C01815=1065.193,415.285,383.687,175.579,36.944,156.981
C01816=1065.183,414.985,383.742,175.571,36.933,156.978
C01817=1065.173,414.684,383.796,175.562,36.921,156.975
C01818=1065.163,414.383,383.850,175.554,36.909,156.972
C01819=1065.153,414.082,383.904,175.545,36.897,156.969
C01820=1065.144,413.837,383.948,175.539,36.887,156.967
C01821=1065.136,413.591,383.993,175.532,36.878,156.964
C01822=1065.128,413.345,384.036,175.525,36.869,156.962
C01823=1065.120,413.099,384.080,175.519,36.859,156.960
C01824=1065.111,412.853,384.125,175.511,36.850,156.957
C01825=1065.103,412.606,384.168,175.505,36.840,156.955
C01826=1065.095,412.361,384.213,175.498,36.831,156.952
C01827=1065.086,412.115,384.256,175.492,36.822,156.950
C01828=1065.079,411.869,384.300,175.485,36.812,156.948
C01829=1065.071,411.623,384.344,175.479,36.803,156.945
C01830=1065.063,411.377,384.388,175.472,36.794,156.943
C01831=1065.054,411.131,384.432,175.466,36.784,156.941
C01832=1065.046,410.885,384.475,175.459,36.775,156.938
C01833=1065.039,410.639,384.519,175.452,36.766,156.936
C01834=1065.030,410.393,384.563,175.445,36.756,156.934
C01835=1065.022,410.147,384.606,175.439,36.747,156.931
C01836=1065.014,409.900,384.650,175.432,36.738,156.929
C01837=1065.006,409.654,384.693,175.426,36.729,156.927
C01838=1064.998,409.409,384.737,175.420,36.720,156.924
C01839=1064.991,409.163,384.780,175.413,36.711,156.922
C01840=1064.983,408.917,384.824,175.407,36.702,156.920
C01841=1064.974,408.671,384.867,175.400,36.693,156.918
C01842=1064.966,408.424,384.911,175.394,36.684,156.915
C01843=1064.959,408.178,384.954,175.388,36.675,156.913
C01844=1064.951,407.932,384.997,175.381,36.666,156.911
C01845=1064.943,407.686,385.041,175.376,36.657,156.909
C01846=1064.935,407.440,385.084,175.369,36.648,156.906
C01847=1064.927,407.194,385.127,175.363,36.639,156.904
C01848=1064.920,406.948,385.171,175.357,36.630,156.902
C01849=1064.912,406.702,385.214,175.350,36.621,156.900
C01850=1064.903,406.456,385.257,175.344,36.613,156.898
C01851=1064.896,406.210,385.300,175.338,36.603,156.895
C01852=1064.888,405.963,385.343,175.331,36.595,156.893
C01853=1064.880,405.717,385.386,175.325,36.586,156.891
C01854=1064.872,405.471,385.429,175.320,36.577,156.889
C01855=1064.865,405.225,385.472,175.313,36.568,156.887
C01856=1064.856,404.978,385.515,175.307,36.560,156.885
C01857=1064.850,404.732,385.558,175.301,36.551,156.882
C01858=1064.841,404.486,385.601,175.295,36.543,156.880
C01859=1064.833,404.240,385.644,175.288,36.534,156.878
C01860=1064.826,403.994,385.686,175.283,36.525,156.876
C01861=1064.817,403.748,385.729,175.277,36.517,156.874
C01862=1064.810,403.501,385.772,175.270,36.508,156.872
C01863=1064.802,403.255,385.814,175.264,36.500,156.870
C01864=1064.794,403.009,385.857,175.258,36.492,156.868
C01865=1064.787,402.762,385.900,175.253,36.483,156.866
C01866=1064.779,402.516,385.941,175.247,36.474,156.863
C01867=1064.771,402.270,385.985,175.240,36.466,156.861
C01868=1064.763,402.023,386.027,175.234,36.458,156.859
C01869=1064.756,401.777,386.069,175.229,36.449,156.857
C01870=1064.748,401.531,386.111,175.223,36.441,156.855
C01871=1064.740,401.285,386.154,175.217,36.433,156.853
C01872=1064.730,400.989,386.205,175.210,36.422,156.851
C01873=1064.721,400.693,386.256,175.203,36.413,156.848
C01874=1064.712,400.397,386.307,175.195,36.403,156.846
C01875=1064.703,400.101,386.357,175.189,36.393,156.843
C01876=1064.695,399.854,386.400,175.183,36.385,156.841
C01877=1064.688,399.608,386.441,175.177,36.376,156.839
C01878=1064.680,399.362,386.483,175.171,36.368,156.838
C01879=1064.672,399.116,386.526,175.165,36.360,156.836
C01880=1064.664,398.870,386.568,175.159,36.352,156.834
C01881=1064.657,398.624,386.610,175.154,36.344,156.832
C01882=1064.649,398.377,386.653,175.148,36.336,156.830
C01883=1064.642,398.130,386.694,175.143,36.328,156.828
C01884=1064.634,397.884,386.736,175.137,36.320,156.826
C01885=1064.627,397.638,386.778,175.131,36.312,156.824
C01886=1064.619,397.391,386.819,175.125,36.304,156.822
C01887=1064.611,397.145,386.861,175.119,36.296,156.820
C01888=1064.604,396.899,386.903,175.114,36.288,156.818
C01889=1064.596,396.652,386.944,175.108,36.280,156.816
C01890=1064.589,396.406,386.986,175.103,36.272,156.814
C01891=1064.581,396.160,387.028,175.097,36.264,156.812
C01892=1064.573,395.913,387.070,175.091,36.256,156.810
C01893=1064.566,395.667,387.112,175.086,36.248,156.808
C01894=1064.558,395.421,387.152,175.080,36.241,156.807
C01895=1064.550,395.174,387.194,175.075,36.233,156.805
C01896=1064.543,394.928,387.236,175.069,36.225,156.803
C01897=1064.536,394.682,387.277,175.064,36.217,156.801
C01898=1064.528,394.436,387.319,175.058,36.209,156.799
C01899=1064.521,394.189,387.360,175.053,36.202,156.797
C01900=1064.513,393.943,387.401,175.047,36.194,156.795
C01901=1064.506,393.697,387.443,175.042,36.186,156.793
C01902=1064.498,393.450,387.484,175.036,36.179,156.792
C01903=1064.490,393.204,387.525,175.031,36.171,156.790
C01904=1064.483,392.957,387.566,175.025,36.163,156.788
C01905=1064.476,392.711,387.607,175.020,36.156,156.786
C01906=1064.468,392.465,387.649,175.014,36.148,156.784
C01907=1064.460,392.218,387.690,175.009,36.141,156.782
C01908=1064.453,391.972,387.731,175.003,36.133,156.781
C01909=1064.446,391.725,387.773,174.998,36.125,156.779
C01910=1064.438,391.479,387.813,174.992,36.118,156.777
C01911=1064.430,391.232,387.854,174.987,36.110,156.775
C01912=1064.424,390.986,387.895,174.982,36.103,156.773
C01913=1064.416,390.740,387.936,174.976,36.095,156.772
C01914=1064.408,390.493,387.977,174.971,36.088,156.770
C01915=1064.401,390.247,388.018,174.965,36.080,156.768
C01916=1064.393,390.000,388.058,174.960,36.073,156.766
C01917=1064.386,389.753,388.099,174.954,36.066,156.765
C01918=1064.378,389.507,388.140,174.949,36.058,156.763
C01919=1064.371,389.261,388.181,174.944,36.051,156.761
C01920=1064.364,389.014,388.221,174.938,36.044,156.759
C01921=1064.356,388.768,388.262,174.933,36.037,156.758
C01922=1064.348,388.521,388.303,174.929,36.029,156.756
C01923=1064.341,388.274,388.343,174.923,36.022,156.754
C01924=1064.334,388.029,388.384,174.918,36.015,156.752
C01925=1064.326,387.782,388.424,174.912,36.007,156.751
C01926=1064.319,387.535,388.465,174.907,36.000,156.749
C01927=1064.311,387.289,388.505,174.902,35.993,156.747
C01928=1064.303,387.010,388.551,174.896,35.985,156.745
C01929=1064.295,386.730,388.597,174.890,35.977,156.743
C01930=1064.286,386.451,388.643,174.884,35.968,156.742
C01931=1064.278,386.171,388.689,174.878,35.961,156.740
C01932=1064.271,385.924,388.729,174.873,35.954,156.738
C01933=1064.264,385.677,388.769,174.868,35.946,156.736
C01934=1064.256,385.431,388.810,174.862,35.939,156.735
C01935=1064.249,385.185,388.849,174.858,35.932,156.733
C01936=1064.242,384.938,388.890,174.853,35.925,156.731
C01937=1064.234,384.692,388.930,174.847,35.918,156.730
C01938=1064.227,384.445,388.970,174.842,35.911,156.728
C01939=1064.220,384.198,389.011,174.837,35.904,156.726
C01940=1064.212,383.952,389.050,174.832,35.897,156.725
C01941=1064.205,383.704,389.091,174.827,35.890,156.723
C01942=1064.198,383.459,389.131,174.822,35.883,156.721
C01943=1064.190,383.212,389.171,174.817,35.876,156.720
C01944=1064.184,382.965,389.211,174.812,35.869,156.718
C01945=1064.176,382.718,389.251,174.807,35.862,156.717
C01946=1064.169,382.472,389.290,174.801,35.855,156.715
C01947=1064.162,382.225,389.331,174.797,35.848,156.713
C01948=1064.155,381.979,389.371,174.792,35.841,156.712
C01949=1064.147,381.732,389.410,174.787,35.834,156.710
C01950=1064.141,381.485,389.451,174.782,35.827,156.708
C01951=1064.134,381.239,389.490,174.776,35.821,156.707
C01952=1064.126,380.992,389.530,174.772,35.814,156.705
C01953=1064.119,380.746,389.569,174.767,35.807,156.704
C01954=1064.112,380.498,389.609,174.762,35.800,156.702
C01955=1064.105,380.252,389.649,174.757,35.794,156.701
C01956=1064.097,380.005,389.689,174.753,35.787,156.699
C01957=1064.090,379.759,389.728,174.747,35.780,156.697
C01958=1064.083,379.511,389.768,174.742,35.774,156.696
C01959=1064.076,379.265,389.807,174.737,35.767,156.694
C01960=1064.069,379.019,389.847,174.733,35.760,156.693
C01961=1064.061,378.772,389.886,174.728,35.754,156.691
C01962=1064.054,378.525,389.926,174.723,35.747,156.690
C01963=1064.047,378.278,389.965,174.718,35.740,156.688
C01964=1064.040,378.032,390.004,174.713,35.734,156.687
C01965=1064.033,377.785,390.043,174.708,35.727,156.685
C01966=1064.025,377.538,390.083,174.703,35.720,156.684
C01967=1064.018,377.291,390.122,174.698,35.714,156.682
C01968=1064.011,377.045,390.161,174.694,35.707,156.680
C01969=1064.004,376.798,390.200,174.689,35.701,156.679
C01970=1063.997,376.551,390.240,174.684,35.694,156.678
C01971=1063.990,376.304,390.279,174.680,35.688,156.676
C01972=1063.983,376.058,390.319,174.675,35.681,156.674
C01973=1063.976,375.811,390.357,174.670,35.675,156.673
C01974=1063.968,375.564,390.397,174.665,35.668,156.672
C01975=1063.961,375.318,390.436,174.660,35.661,156.670
C01976=1063.955,375.071,390.475,174.655,35.655,156.669
C01977=1063.948,374.824,390.514,174.650,35.649,156.667
C01978=1063.941,374.577,390.553,174.646,35.642,156.666
C01979=1063.933,374.330,390.592,174.641,35.636,156.664
C01980=1063.926,374.083,390.631,174.636,35.630,156.663
C01981=1063.919,373.837,390.670,174.632,35.623,156.661
C01982=1063.912,373.590,390.708,174.627,35.617,156.660
C01983=1063.905,373.343,390.747,174.622,35.610,156.658
C01984=1063.898,373.094,390.787,174.618,35.604,156.657
C01985=1063.892,372.845,390.826,174.613,35.597,156.655
C01986=1063.884,372.597,390.865,174.608,35.591,156.654
C01987=1063.877,372.347,390.904,174.604,35.584,156.652
C01988=1063.870,372.101,390.943,174.599,35.578,156.651
C01989=1063.863,371.854,390.981,174.594,35.572,156.650
C01990=1063.856,371.607,391.020,174.590,35.566,156.648
C01991=1063.849,371.360,391.059,174.585,35.560,156.647
C01992=1063.841,371.113,391.098,174.580,35.554,156.645
C01993=1063.835,370.866,391.136,174.576,35.548,156.644
C01994=1063.827,370.619,391.174,174.571,35.541,156.643
C01995=1063.820,370.372,391.213,174.566,35.535,156.641
C01996=1063.813,370.126,391.252,174.562,35.529,156.640
C01997=1063.806,369.878,391.289,174.557,35.522,156.638
C01998=1063.799,369.632,391.328,174.553,35.517,156.637
C01999=1063.792,369.385,391.367,174.549,35.511,156.635
C02000=1063.785,369.138,391.405,174.544,35.504,156.634
C02001=1063.778,368.891,391.443,174.540,35.498,156.633
C02002=1063.771,368.644,391.481,174.535,35.492,156.631
C02003=1063.764,368.397,391.520,174.530,35.486,156.630
C02004=1063.758,368.150,391.558,174.526,35.480,156.629
C02005=1063.750,367.904,391.597,174.521,35.474,156.627
C02006=1063.744,367.656,391.635,174.517,35.468,156.626
C02007=1063.736,367.410,391.673,174.512,35.462,156.624
C02008=1063.730,367.163,391.711,174.507,35.456,156.623
C02009=1063.723,366.916,391.750,174.503,35.449,156.622
C02010=1063.716,366.669,391.787,174.499,35.443,156.620
C02011=1063.710,366.421,391.825,174.495,35.438,156.619
C02012=1063.702,366.175,391.863,174.490,35.431,156.618
C02013=1063.695,365.928,391.902,174.485,35.425,156.616
C02014=1063.688,365.681,391.940,174.481,35.420,156.615
C02015=1063.682,365.434,391.978,174.476,35.413,156.614
C02016=1063.675,365.187,392.015,174.472,35.408,156.612
C02017=1063.668,364.940,392.054,174.468,35.402,156.611
C02018=1063.661,364.693,392.092,174.464,35.395,156.609
C02019=1063.654,364.446,392.130,174.459,35.390,156.608
C02020=1063.648,364.199,392.167,174.454,35.384,156.607
C02021=1063.641,363.952,392.205,174.450,35.378,156.606
C02022=1063.633,363.705,392.243,174.445,35.372,156.604
C02023=1063.627,363.458,392.281,174.442,35.366,156.603
C02024=1063.620,363.211,392.319,174.437,35.361,156.602
C02025=1063.612,362.964,392.356,174.433,35.355,156.600
C02026=1063.607,362.717,392.394,174.428,35.349,156.599
C02027=1063.599,362.470,392.432,174.424,35.343,156.598
C02028=1063.592,362.223,392.469,174.419,35.337,156.596
C02029=1063.585,361.975,392.507,174.416,35.332,156.595
C02030=1063.579,361.729,392.544,174.411,35.326,156.594
C02031=1063.572,361.482,392.582,174.406,35.320,156.593
C02032=1063.564,361.234,392.619,174.402,35.314,156.591
C02033=1063.557,360.987,392.657,174.398,35.309,156.590
C02034=1063.551,360.741,392.695,174.394,35.303,156.589
C02035=1063.544,360.493,392.732,174.389,35.297,156.588
C02036=1063.538,360.254,392.768,174.385,35.292,156.586
C02037=1063.531,360.015,392.804,174.381,35.286,156.585
C02038=1063.524,359.776,392.840,174.377,35.280,156.584
C02039=1063.518,359.537,392.876,174.372,35.275,156.583
C02040=1063.511,359.298,392.912,174.369,35.270,156.581
C02041=1063.505,359.059,392.949,174.364,35.264,156.580
C02042=1063.498,358.820,392.985,174.361,35.259,156.579
C02043=1063.491,358.581,393.021,174.356,35.253,156.578
C02044=1063.485,358.334,393.058,174.352,35.247,156.576
C02045=1063.478,358.087,393.095,174.348,35.242,156.575
C02046=1063.471,357.840,393.133,174.344,35.236,156.574
C02047=1063.464,357.592,393.169,174.339,35.230,156.573
C02048=1063.457,357.345,393.207,174.335,35.225,156.572
C02049=1063.451,357.098,393.243,174.331,35.220,156.570
C02050=1063.443,356.851,393.281,174.327,35.214,156.569
C02051=1063.437,356.604,393.317,174.322,35.208,156.568
C02052=1063.430,356.357,393.355,174.319,35.203,156.567
C02053=1063.423,356.109,393.392,174.314,35.198,156.565
C02054=1063.416,355.863,393.429,174.310,35.192,156.564
C02055=1063.409,355.615,393.466,174.305,35.186,156.563
C02056=1063.403,355.368,393.502,174.302,35.181,156.562
C02057=1063.396,355.121,393.540,174.297,35.175,156.560
C02058=1063.389,354.874,393.576,174.293,35.170,156.559
C02059=1063.382,354.627,393.614,174.290,35.165,156.558
C02060=1063.376,354.380,393.650,174.285,35.159,156.557
C02061=1063.369,354.132,393.687,174.281,35.154,156.556
C02062=1063.362,353.885,393.723,174.277,35.148,156.554
C02063=1063.356,353.638,393.760,174.273,35.142,156.553
C02064=1063.349,353.391,393.797,174.269,35.137,156.552
C02065=1063.343,353.143,393.834,174.265,35.132,156.551
C02066=1063.336,352.896,393.871,174.260,35.126,156.550
C02067=1063.329,352.649,393.908,174.257,35.121,156.548
C02068=1063.323,352.402,393.944,174.252,35.116,156.547
C02069=1063.316,352.154,393.981,174.248,35.110,156.546
C02070=1063.309,351.907,394.017,174.244,35.105,156.545
C02071=1063.302,351.660,394.054,174.240,35.100,156.544
C02072=1063.295,351.413,394.090,174.237,35.094,156.543
C02073=1063.289,351.166,394.127,174.232,35.089,156.541
C02074=1063.282,350.918,394.163,174.228,35.084,156.540
C02075=1063.276,350.671,394.200,174.224,35.078,156.539
C02076=1063.268,350.424,394.236,174.220,35.073,156.538
C02077=1063.262,350.177,394.272,174.216,35.068,156.537
C02078=1063.255,349.929,394.309,174.212,35.062,156.536
C02079=1063.248,349.682,394.345,174.207,35.057,156.535
C02080=1063.241,349.435,394.382,174.204,35.052,156.533
C02081=1063.235,349.188,394.418,174.200,35.046,156.532
C02082=1063.228,348.940,394.455,174.196,35.041,156.531
C02083=1063.221,348.693,394.490,174.192,35.036,156.530
C02084=1063.215,348.446,394.526,174.187,35.030,156.529
C02085=1063.208,348.198,394.563,174.184,35.025,156.528
C02086=1063.201,347.951,394.599,174.180,35.020,156.527
C02087=1063.195,347.704,394.635,174.176,35.015,156.525
C02088=1063.189,347.457,394.671,174.172,35.010,156.524
C02089=1063.181,347.209,394.707,174.168,35.005,156.523
C02090=1063.175,346.962,394.744,174.164,35.000,156.522
C02091=1063.169,346.714,394.780,174.161,34.994,156.521
C02092=1063.162,346.478,394.814,174.156,34.989,156.520
C02093=1063.156,346.241,394.848,174.153,34.984,156.519
C02094=1063.150,346.004,394.883,174.149,34.979,156.518
C02095=1063.143,345.767,394.917,174.145,34.974,156.517
C02096=1063.137,345.530,394.952,174.142,34.970,156.516
C02097=1063.130,345.293,394.987,174.137,34.965,156.515
C02098=1063.124,345.056,395.021,174.134,34.959,156.513
C02099=1063.117,344.819,395.056,174.130,34.955,156.512
C02100=1063.111,344.572,395.091,174.126,34.950,156.511
C02101=1063.104,344.324,395.127,174.123,34.944,156.510
C02102=1063.098,344.077,395.163,174.118,34.939,156.509
C02103=1063.091,343.830,395.199,174.115,34.934,156.508
C02104=1063.085,343.582,395.235,174.110,34.929,156.507
C02105=1063.078,343.334,395.270,174.107,34.924,156.506
C02106=1063.071,343.088,395.306,174.103,34.919,156.505
C02107=1063.065,342.840,395.342,174.099,34.914,156.504
C02108=1063.058,342.593,395.377,174.095,34.909,156.503
C02109=1063.052,342.345,395.413,174.092,34.904,156.501
C02110=1063.045,342.098,395.449,174.087,34.899,156.500
C02111=1063.038,341.851,395.484,174.084,34.894,156.499
C02112=1063.032,341.603,395.519,174.080,34.889,156.498
C02113=1063.025,341.356,395.555,174.076,34.884,156.497
C02114=1063.018,341.108,395.591,174.073,34.879,156.496
C02115=1063.012,340.861,395.627,174.068,34.874,156.495
C02116=1063.005,340.613,395.662,174.065,34.869,156.494
C02117=1062.998,340.366,395.697,174.061,34.864,156.493
C02118=1062.992,340.118,395.733,174.057,34.859,156.492
C02119=1062.985,339.871,395.768,174.053,34.854,156.491
C02120=1062.978,339.624,395.803,174.050,34.849,156.490
C02121=1062.972,339.376,395.839,174.046,34.844,156.489
C02122=1062.965,339.129,395.874,174.042,34.840,156.488
C02123=1062.959,338.882,395.909,174.038,34.834,156.487
C02124=1062.953,338.634,395.945,174.034,34.830,156.486
C02125=1062.946,338.387,395.980,174.031,34.825,156.484
C02126=1062.939,338.139,396.015,174.027,34.820,156.483
C02127=1062.932,337.892,396.051,174.023,34.815,156.482
C02128=1062.927,337.645,396.086,174.020,34.810,156.481
C02129=1062.920,337.398,396.121,174.015,34.805,156.480
C02130=1062.913,337.150,396.156,174.012,34.800,156.479
C02131=1062.907,336.902,396.191,174.009,34.795,156.478
C02132=1062.901,336.655,396.226,174.004,34.791,156.477
C02133=1062.894,336.407,396.262,174.001,34.785,156.476
C02134=1062.887,336.160,396.297,173.998,34.781,156.475
C02135=1062.881,335.912,396.332,173.993,34.776,156.474
C02136=1062.874,335.664,396.366,173.990,34.771,156.473
C02137=1062.867,335.417,396.401,173.987,34.766,156.472
C02138=1062.861,335.170,396.436,173.982,34.762,156.471
C02139=1062.854,334.922,396.472,173.979,34.757,156.470
C02140=1062.848,334.675,396.506,173.975,34.752,156.469
C02141=1062.841,334.428,396.541,173.971,34.747,156.468
C02142=1062.834,334.180,396.576,173.968,34.742,156.467
C02143=1062.828,333.932,396.610,173.964,34.738,156.466
C02144=1062.821,333.685,396.646,173.960,34.733,156.465
C02145=1062.814,333.438,396.681,173.957,34.728,156.464
C02146=1062.809,333.189,396.716,173.953,34.723,156.463
C02147=1062.802,332.943,396.750,173.949,34.719,156.462
C02148=1062.795,332.703,396.784,173.946,34.714,156.461
C02149=1062.789,332.464,396.817,173.943,34.709,156.460
C02150=1062.783,332.224,396.851,173.940,34.705,156.459
C02151=1062.777,331.985,396.884,173.935,34.700,156.458
C02152=1062.771,331.746,396.918,173.932,34.695,156.457
C02153=1062.764,331.506,396.951,173.929,34.691,156.456
C02154=1062.758,331.267,396.985,173.925,34.686,156.455
C02155=1062.752,331.028,397.019,173.922,34.682,156.454
C02156=1062.746,330.780,397.053,173.918,34.677,156.453
C02157=1062.739,330.533,397.088,173.914,34.672,156.452
C02158=1062.732,330.285,397.122,173.911,34.668,156.451
C02159=1062.725,330.037,397.156,173.907,34.663,156.450
C02160=1062.720,329.790,397.191,173.904,34.659,156.449
C02161=1062.712,329.543,397.225,173.900,34.654,156.448
C02162=1062.706,329.295,397.259,173.897,34.650,156.447
C02163=1062.699,329.047,397.294,173.893,34.645,156.446
C02164=1062.693,328.800,397.327,173.889,34.640,156.445
C02165=1062.686,328.553,397.362,173.886,34.636,156.444
C02166=1062.679,328.305,397.397,173.883,34.631,156.444
C02167=1062.672,328.057,397.431,173.879,34.627,156.443
C02168=1062.666,327.810,397.465,173.875,34.622,156.442
C02169=1062.660,327.562,397.499,173.872,34.617,156.441
C02170=1062.653,327.314,397.533,173.868,34.613,156.440
C02171=1062.646,327.067,397.568,173.864,34.608,156.439
C02172=1062.639,326.820,397.602,173.861,34.604,156.438
C02173=1062.633,326.572,397.636,173.858,34.599,156.437
C02174=1062.627,326.324,397.670,173.855,34.595,156.436
C02175=1062.620,326.077,397.704,173.850,34.590,156.435
C02176=1062.613,325.829,397.738,173.847,34.585,156.434
C02177=1062.607,325.581,397.772,173.844,34.581,156.433
C02178=1062.600,325.334,397.806,173.840,34.577,156.432
C02179=1062.594,325.086,397.841,173.836,34.572,156.431
C02180=1062.587,324.839,397.874,173.833,34.567,156.430
C02181=1062.581,324.591,397.909,173.830,34.563,156.429
C02182=1062.575,324.344,397.943,173.826,34.559,156.428
C02183=1062.568,324.096,397.976,173.823,34.554,156.427
C02184=1062.562,323.848,398.010,173.819,34.550,156.427
C02185=1062.555,323.600,398.044,173.816,34.545,156.426
C02186=1062.548,323.352,398.078,173.812,34.540,156.425
C02187=1062.542,323.105,398.111,173.809,34.536,156.424
C02188=1062.535,322.857,398.146,173.806,34.532,156.423
C02189=1062.530,322.610,398.180,173.801,34.527,156.422
C02190=1062.523,322.362,398.213,173.798,34.522,156.421
C02191=1062.517,322.114,398.247,173.795,34.518,156.420
C02192=1062.510,321.867,398.281,173.792,34.513,156.419
C02193=1062.504,321.619,398.315,173.788,34.509,156.418
C02194=1062.497,321.372,398.348,173.785,34.505,156.417
C02195=1062.491,321.124,398.382,173.782,34.500,156.416
C02196=1062.484,320.877,398.416,173.778,34.496,156.415
C02197=1062.478,320.629,398.450,173.774,34.491,156.414
C02198=1062.472,320.381,398.483,173.771,34.486,156.413
C02199=1062.465,320.133,398.517,173.768,34.482,156.413
C02200=1062.459,319.886,398.550,173.765,34.478,156.412
C02201=1062.453,319.639,398.584,173.761,34.473,156.411
C02202=1062.446,319.391,398.618,173.758,34.469,156.410
C02203=1062.440,319.143,398.651,173.755,34.464,156.409
C02204=1062.434,318.901,398.684,173.751,34.460,156.408
C02205=1062.428,318.659,398.717,173.747,34.455,156.407
C02206=1062.421,318.416,398.750,173.744,34.451,156.406
C02207=1062.415,318.174,398.783,173.741,34.447,156.405
C02208=1062.409,317.932,398.815,173.738,34.442,156.404
C02209=1062.403,317.690,398.849,173.734,34.438,156.404
C02210=1062.397,317.448,398.881,173.731,34.434,156.403
C02211=1062.391,317.205,398.913,173.728,34.430,156.402
C02212=1062.385,316.958,398.947,173.725,34.425,156.401
C02213=1062.378,316.710,398.980,173.721,34.421,156.400
C02214=1062.372,316.462,399.014,173.718,34.416,156.399
C02215=1062.366,316.215,399.047,173.715,34.412,156.398
C02216=1062.360,315.967,399.081,173.712,34.407,156.397
C02217=1062.353,315.719,399.114,173.708,34.403,156.396
C02218=1062.347,315.471,399.148,173.705,34.398,156.395
C02219=1062.341,315.224,399.180,173.702,34.394,156.394
C02220=1062.334,314.977,399.214,173.699,34.390,156.394
C02221=1062.329,314.729,399.247,173.696,34.386,156.393
C02222=1062.322,314.481,399.280,173.692,34.381,156.392
C02223=1062.316,314.233,399.314,173.689,34.377,156.391
C02224=1062.310,313.986,399.347,173.685,34.372,156.390
C02225=1062.304,313.738,399.380,173.682,34.368,156.389
C02226=1062.297,313.490,399.413,173.678,34.364,156.388
C02227=1062.290,313.242,399.446,173.675,34.360,156.387
C02228=1062.284,313.015,399.476,173.672,34.355,156.387
C02229=1062.279,312.790,399.506,173.670,34.352,156.386
C02230=1062.273,312.563,399.536,173.667,34.348,156.385
C02231=1062.267,312.336,399.566,173.663,34.344,156.384
C02232=1062.260,312.110,399.597,173.660,34.340,156.383
C02233=1062.255,311.884,399.626,173.657,34.336,156.383
C02234=1062.249,311.657,399.656,173.655,34.332,156.382
C02235=1062.243,311.431,399.686,173.652,34.328,156.381
C02236=1062.237,311.183,399.719,173.648,34.324,156.380
C02237=1062.230,310.936,399.752,173.645,34.320,156.379
C02238=1062.224,310.688,399.785,173.642,34.316,156.378
C02239=1062.217,310.441,399.817,173.639,34.312,156.378
C02240=1062.210,310.192,399.850,173.636,34.308,156.377
C02241=1062.204,309.945,399.883,173.632,34.303,156.376
C02242=1062.197,309.697,399.915,173.629,34.299,156.375
C02243=1062.191,309.450,399.948,173.626,34.295,156.374
C02244=1062.185,309.202,399.981,173.623,34.290,156.373
C02245=1062.179,308.954,400.014,173.619,34.286,156.372
C02246=1062.172,308.705,400.046,173.616,34.282,156.372
C02247=1062.166,308.458,400.079,173.613,34.278,156.371
C02248=1062.159,308.210,400.111,173.610,34.274,156.370
C02249=1062.152,307.963,400.144,173.607,34.270,156.369
C02250=1062.146,307.715,400.176,173.603,34.266,156.368
C02251=1062.140,307.467,400.208,173.600,34.261,156.367
C02252=1062.134,307.220,400.241,173.597,34.257,156.366
C02253=1062.128,306.972,400.274,173.594,34.253,156.366
C02254=1062.121,306.724,400.307,173.591,34.248,156.365
C02255=1062.115,306.476,400.339,173.587,34.244,156.364
C02256=1062.108,306.229,400.371,173.584,34.240,156.363
C02257=1062.102,305.981,400.403,173.581,34.236,156.362
C02258=1062.096,305.733,400.435,173.578,34.232,156.361
C02259=1062.090,305.486,400.468,173.575,34.228,156.361
C02260=1062.083,305.238,400.501,173.571,34.224,156.360
C02261=1062.077,304.990,400.533,173.568,34.219,156.359
C02262=1062.070,304.742,400.565,173.565,34.215,156.358
C02263=1062.064,304.495,400.598,173.562,34.211,156.357
C02264=1062.057,304.219,400.634,173.559,34.206,156.356
C02265=1062.051,303.943,400.669,173.554,34.202,156.355
C02266=1062.043,303.667,400.705,173.551,34.197,156.354
C02267=1062.036,303.392,400.741,173.548,34.192,156.353
C02268=1062.030,303.144,400.774,173.545,34.188,156.353
C02269=1062.024,302.896,400.806,173.542,34.184,156.352
C02270=1062.017,302.649,400.838,173.538,34.180,156.351
C02271=1062.011,302.401,400.870,173.535,34.175,156.350
C02272=1062.005,302.153,400.903,173.532,34.171,156.349
C02273=1061.999,301.905,400.935,173.529,34.167,156.348
C02274=1061.993,301.658,400.967,173.526,34.163,156.348
C02275=1061.986,301.410,400.999,173.524,34.159,156.347
C02276=1061.980,301.162,401.031,173.520,34.155,156.346
C02277=1061.974,300.914,401.063,173.517,34.151,156.345
C02278=1061.968,300.666,401.095,173.514,34.146,156.344
C02279=1061.961,300.418,401.127,173.511,34.142,156.343
C02280=1061.955,300.171,401.160,173.508,34.138,156.343
C02281=1061.950,299.923,401.191,173.504,34.134,156.342
C02282=1061.944,299.675,401.223,173.501,34.130,156.341
C02283=1061.937,299.428,401.255,173.499,34.126,156.340
C02284=1061.931,299.179,401.288,173.496,34.121,156.339
C02285=1061.925,298.931,401.320,173.493,34.117,156.338
C02286=1061.919,298.684,401.351,173.490,34.113,156.338
C02287=1061.912,298.436,401.383,173.486,34.109,156.337
C02288=1061.906,298.188,401.415,173.483,34.105,156.336
C02289=1061.900,297.940,401.447,173.480,34.101,156.335
C02290=1061.895,297.693,401.479,173.478,34.096,156.334
C02291=1061.888,297.445,401.510,173.475,34.092,156.333
C02292=1061.882,297.197,401.543,173.472,34.088,156.333
C02293=1061.876,296.949,401.575,173.468,34.084,156.332
C02294=1061.869,296.701,401.607,173.465,34.080,156.331
C02295=1061.864,296.453,401.638,173.462,34.076,156.330
C02296=1061.857,296.205,401.670,173.459,34.072,156.329
C02297=1061.851,295.957,401.702,173.457,34.068,156.328
C02298=1061.844,295.709,401.733,173.454,34.064,156.328
C02299=1061.838,295.462,401.764,173.450,34.060,156.327
C02300=1061.832,295.214,401.796,173.447,34.056,156.326
C02301=1061.826,294.966,401.828,173.444,34.052,156.325
C02302=1061.820,294.718,401.860,173.441,34.048,156.324
C02303=1061.813,294.471,401.891,173.439,34.043,156.324
C02304=1061.807,294.223,401.922,173.436,34.040,156.323
C02305=1061.801,293.974,401.954,173.432,34.036,156.322
C02306=1061.794,293.726,401.985,173.429,34.031,156.321
C02307=1061.788,293.479,402.016,173.426,34.027,156.320
C02308=1061.782,293.231,402.048,173.424,34.024,156.320
C02309=1061.776,292.983,402.080,173.421,34.020,156.319
C02310=1061.769,292.735,402.111,173.418,34.015,156.318
C02311=1061.763,292.487,402.143,173.415,34.011,156.317
C02312=1061.757,292.239,402.173,173.411,34.008,156.317
C02313=1061.750,291.991,402.205,173.408,34.003,156.316
C02314=1061.745,291.743,402.236,173.406,33.999,156.315
C02315=1061.738,291.495,402.268,173.403,33.996,156.314
C02316=1061.733,291.262,402.297,173.400,33.991,156.313
C02317=1061.726,291.030,402.326,173.398,33.988,156.313
C02318=1061.721,290.797,402.356,173.395,33.984,156.312
C02319=1061.714,290.564,402.385,173.391,33.980,156.311
C02320=1061.709,290.331,402.414,173.389,33.976,156.310
C02321=1061.703,290.099,402.443,173.386,33.973,156.310
C02322=1061.697,289.866,402.473,173.384,33.969,156.309
C02323=1061.691,289.634,402.502,173.381,33.965,156.308
C02324=1061.685,289.385,402.533,173.378,33.961,156.307
C02325=1061.679,289.138,402.564,173.376,33.957,156.307
C02326=1061.673,288.889,402.595,173.372,33.953,156.306
C02327=1061.667,288.642,402.626,173.369,33.950,156.305
C02328=1061.661,288.394,402.658,173.366,33.945,156.304
C02329=1061.654,288.146,402.689,173.363,33.941,156.303
C02330=1061.648,287.898,402.720,173.361,33.938,156.303
C02331=1061.642,287.650,402.751,173.358,33.933,156.302
C02332=1061.635,287.401,402.781,173.355,33.930,156.301
C02333=1061.629,287.154,402.812,173.351,33.926,156.300
C02334=1061.623,286.906,402.843,173.349,33.921,156.299
C02335=1061.617,286.658,402.874,173.346,33.918,156.299
C02336=1061.610,286.410,402.905,173.343,33.914,156.298
C02337=1061.603,286.162,402.936,173.341,33.910,156.297
C02338=1061.598,285.914,402.967,173.338,33.906,156.296
C02339=1061.591,285.666,402.997,173.335,33.902,156.296
C02340=1061.585,285.418,403.029,173.331,33.898,156.295
C02341=1061.579,285.170,403.059,173.329,33.894,156.294
C02342=1061.573,284.922,403.090,173.326,33.890,156.293
C02343=1061.566,284.674,403.121,173.323,33.886,156.293
C02344=1061.560,284.426,403.151,173.320,33.882,156.292
C02345=1061.554,284.178,403.182,173.318,33.878,156.291
C02346=1061.548,283.931,403.213,173.315,33.874,156.290
C02347=1061.541,283.682,403.244,173.312,33.870,156.289
C02348=1061.535,283.434,403.274,173.309,33.866,156.289
C02349=1061.529,283.186,403.305,173.306,33.863,156.288
C02350=1061.523,282.939,403.336,173.303,33.858,156.287
C02351=1061.516,282.690,403.367,173.301,33.855,156.286
C02352=1061.511,282.442,403.397,173.298,33.851,156.286
C02353=1061.504,282.194,403.428,173.295,33.846,156.285
C02354=1061.498,281.946,403.458,173.293,33.843,156.284
C02355=1061.492,281.697,403.489,173.290,33.839,156.283
C02356=1061.486,281.450,403.520,173.286,33.835,156.283
C02357=1061.479,281.202,403.551,173.284,33.831,156.282
C02358=1061.474,280.954,403.581,173.281,33.827,156.281
C02359=1061.468,280.706,403.611,173.278,33.823,156.280
C02360=1061.461,280.458,403.641,173.276,33.819,156.279
C02361=1061.455,280.210,403.672,173.273,33.815,156.279
C02362=1061.448,279.961,403.703,173.270,33.811,156.278
C02363=1061.443,279.714,403.733,173.268,33.807,156.277
C02364=1061.437,279.466,403.763,173.264,33.803,156.276
C02365=1061.430,279.217,403.794,173.261,33.799,156.276
C02366=1061.424,278.970,403.824,173.259,33.795,156.275
C02367=1061.417,278.721,403.854,173.256,33.792,156.274
C02368=1061.412,278.473,403.885,173.253,33.787,156.273
C02369=1061.405,278.225,403.915,173.251,33.784,156.273
C02370=1061.399,277.977,403.945,173.248,33.780,156.272
C02371=1061.393,277.730,403.976,173.245,33.776,156.271
C02372=1061.387,277.502,404.004,173.243,33.772,156.270
C02373=1061.381,277.274,404.030,173.240,33.769,156.270
C02374=1061.376,277.047,404.058,173.237,33.765,156.269
C02375=1061.370,276.819,404.086,173.235,33.762,156.268
C02376=1061.364,276.592,404.114,173.232,33.758,156.267
C02377=1061.359,276.365,404.141,173.230,33.754,156.267
C02378=1061.353,276.138,404.169,173.227,33.751,156.266
C02379=1061.347,275.911,404.197,173.225,33.748,156.265
C02380=1061.342,275.662,404.226,173.222,33.743,156.265
C02381=1061.335,275.414,404.257,173.220,33.740,156.264
C02382=1061.329,275.166,404.287,173.216,33.736,156.263
C02383=1061.323,274.918,404.317,173.214,33.732,156.262
C02384=1061.317,274.669,404.347,173.211,33.728,156.262
C02385=1061.310,274.422,404.377,173.208,33.724,156.261
C02386=1061.304,274.174,404.407,173.206,33.720,156.260
C02387=1061.298,273.925,404.438,173.203,33.716,156.259
C02388=1061.292,273.677,404.467,173.201,33.712,156.259
C02389=1061.286,273.429,404.497,173.198,33.709,156.258
C02390=1061.280,273.181,404.526,173.195,33.705,156.257
C02391=1061.273,272.933,404.557,173.193,33.701,156.256
C02392=1061.267,272.685,404.587,173.189,33.697,156.256
C02393=1061.261,272.437,404.617,173.187,33.693,156.255
C02394=1061.255,272.188,404.647,173.184,33.689,156.254
C02395=1061.248,271.940,404.676,173.182,33.685,156.253
C02396=1061.243,271.692,404.707,173.179,33.681,156.253
C02397=1061.236,271.444,404.736,173.176,33.678,156.252
C02398=1061.230,271.196,404.766,173.174,33.674,156.251
C02399=1061.224,270.948,404.795,173.171,33.670,156.250
C02400=1061.218,270.700,404.826,173.169,33.666,156.250
C02401=1061.212,270.452,404.855,173.166,33.662,156.249
C02402=1061.205,270.204,404.885,173.163,33.658,156.248
C02403=1061.199,269.955,404.915,173.160,33.654,156.247
C02404=1061.192,269.707,404.944,173.158,33.651,156.247
C02405=1061.187,269.459,404.974,173.155,33.647,156.246
C02406=1061.181,269.211,405.003,173.152,33.643,156.245
C02407=1061.175,268.963,405.033,173.150,33.639,156.244
C02408=1061.168,268.714,405.063,173.147,33.635,156.244
C02409=1061.161,268.467,405.093,173.145,33.631,156.243
C02410=1061.156,268.218,405.122,173.142,33.628,156.242
C02411=1061.150,267.970,405.151,173.140,33.623,156.241
C02412=1061.143,267.723,405.181,173.137,33.620,156.241
C02413=1061.137,267.474,405.211,173.134,33.616,156.240
C02414=1061.131,267.225,405.240,173.131,33.612,156.239
C02415=1061.124,266.977,405.269,173.129,33.608,156.238
C02416=1061.119,266.729,405.299,173.126,33.604,156.238
C02417=1061.112,266.481,405.328,173.124,33.600,156.237
C02418=1061.106,266.233,405.357,173.121,33.597,156.236
C02419=1061.100,265.984,405.387,173.118,33.593,156.235
C02420=1061.094,265.736,405.417,173.116,33.589,156.235
C02421=1061.087,265.488,405.446,173.113,33.585,156.234
C02422=1061.082,265.240,405.476,173.111,33.581,156.233
C02423=1061.075,264.992,405.505,173.108,33.577,156.233
C02424=1061.069,264.744,405.534,173.106,33.574,156.232
C02425=1061.063,264.496,405.563,173.102,33.570,156.231
C02426=1061.057,264.247,405.593,173.100,33.566,156.230
C02427=1061.051,263.999,405.622,173.097,33.562,156.230
C02428=1061.045,263.774,405.649,173.095,33.559,156.229
C02429=1061.040,263.548,405.675,173.093,33.555,156.228
C02430=1061.035,263.322,405.702,173.091,33.551,156.228
C02431=1061.028,263.097,405.729,173.088,33.548,156.227
C02432=1061.023,262.872,405.755,173.086,33.545,156.226
C02433=1061.017,262.646,405.782,173.084,33.541,156.226
C02434=1061.011,262.421,405.807,173.082,33.538,156.225
C02435=1061.006,262.195,405.834,173.079,33.534,156.224
C02436=1060.999,261.947,405.863,173.077,33.531,156.224
C02437=1060.993,261.699,405.892,173.074,33.527,156.223
C02438=1060.987,261.451,405.921,173.071,33.523,156.222
C02439=1060.981,261.203,405.950,173.068,33.519,156.221
C02440=1060.974,260.954,405.979,173.066,33.516,156.221
C02441=1060.967,260.706,406.009,173.063,33.511,156.220
C02442=1060.960,260.458,406.037,173.061,33.508,156.219
C02443=1060.955,260.209,406.065,173.059,33.504,156.218
C02444=1060.948,259.961,406.094,173.056,33.500,156.218
C02445=1060.942,259.713,406.123,173.054,33.497,156.217
C02446=1060.936,259.465,406.152,173.051,33.493,156.216
C02447=1060.930,259.217,406.181,173.049,33.489,156.216
C02448=1060.923,258.968,406.210,173.046,33.485,156.215
C02449=1060.917,258.720,406.239,173.044,33.482,156.214
C02450=1060.911,258.472,406.268,173.041,33.477,156.213
C02451=1060.905,258.223,406.297,173.039,33.474,156.213
C02452=1060.899,257.975,406.326,173.035,33.470,156.212
C02453=1060.893,257.727,406.354,173.033,33.466,156.211
C02454=1060.886,257.478,406.383,173.031,33.462,156.210
C02455=1060.879,257.231,406.412,173.028,33.459,156.210
C02456=1060.873,256.982,406.440,173.026,33.455,156.209
C02457=1060.867,256.734,406.469,173.023,33.451,156.208
C02458=1060.861,256.486,406.498,173.021,33.447,156.208
C02459=1060.855,256.237,406.526,173.018,33.443,156.207
C02460=1060.849,255.989,406.556,173.016,33.440,156.206
C02461=1060.843,255.741,406.585,173.014,33.436,156.205
C02462=1060.837,255.492,406.613,173.011,33.432,156.205
C02463=1060.830,255.244,406.642,173.009,33.428,156.204
C02464=1060.823,254.996,406.670,173.006,33.424,156.203
C02465=1060.818,254.748,406.698,173.004,33.420,156.202
C02466=1060.812,254.500,406.727,173.002,33.417,156.202
C02467=1060.806,254.251,406.756,172.998,33.412,156.201
C02468=1060.800,254.003,406.785,172.996,33.409,156.200
C02469=1060.794,253.754,406.813,172.993,33.405,156.200
C02470=1060.787,253.506,406.842,172.991,33.401,156.199
C02471=1060.781,253.257,406.870,172.989,33.397,156.198
C02472=1060.774,253.009,406.899,172.986,33.394,156.197
C02473=1060.769,252.761,406.927,172.984,33.390,156.197
C02474=1060.763,252.513,406.956,172.982,33.386,156.196
C02475=1060.757,252.264,406.984,172.979,33.382,156.195
C02476=1060.751,252.016,407.013,172.977,33.378,156.194
C02477=1060.744,251.768,407.041,172.974,33.374,156.194
C02478=1060.738,251.520,407.070,172.972,33.370,156.193
C02479=1060.732,251.271,407.098,172.970,33.367,156.192
C02480=1060.726,251.023,407.126,172.967,33.363,156.191
C02481=1060.720,250.775,407.155,172.965,33.359,156.191
C02482=1060.714,250.526,407.184,172.963,33.355,156.190
C02483=1060.708,250.278,407.211,172.960,33.351,156.189
C02484=1060.702,250.052,407.238,172.958,33.347,156.189
C02485=1060.697,249.825,407.264,172.955,33.344,156.188
C02486=1060.691,249.598,407.290,172.953,33.341,156.187
C02487=1060.686,249.372,407.316,172.951,33.337,156.187
C02488=1060.680,249.145,407.342,172.949,33.333,156.186
C02489=1060.674,248.919,407.367,172.946,33.330,156.185
C02490=1060.669,248.692,407.393,172.944,33.326,156.185
C02491=1060.664,248.466,407.419,172.942,33.323,156.184
C02492=1060.658,248.218,407.447,172.940,33.319,156.183
C02493=1060.652,247.969,407.475,172.938,33.315,156.182
C02494=1060.645,247.721,407.504,172.935,33.311,156.182
C02495=1060.640,247.473,407.532,172.933,33.307,156.181
C02496=1060.634,247.224,407.560,172.931,33.304,156.180
C02497=1060.628,246.976,407.588,172.928,33.299,156.179
C02498=1060.621,246.727,407.616,172.926,33.296,156.179
C02499=1060.616,246.480,407.645,172.924,33.292,156.178
C02500=1060.610,246.231,407.673,172.921,33.288,156.177
C02501=1060.603,245.982,407.701,172.919,33.284,156.177
C02502=1060.598,245.734,407.729,172.917,33.280,156.176
C02503=1060.592,245.486,407.757,172.915,33.276,156.175
C02504=1060.585,245.237,407.785,172.912,33.273,156.174
C02505=1060.579,244.988,407.813,172.910,33.268,156.174
C02506=1060.573,244.741,407.840,172.908,33.265,156.173
C02507=1060.567,244.492,407.869,172.904,33.261,156.172
C02508=1060.561,244.244,407.896,172.902,33.257,156.171
C02509=1060.555,243.995,407.924,172.900,33.253,156.171
C02510=1060.549,243.747,407.952,172.897,33.249,156.170
C02511=1060.543,243.498,407.980,172.895,33.245,156.169
C02512=1060.537,243.250,408.008,172.893,33.242,156.168
C02513=1060.531,243.002,408.036,172.891,33.238,156.168
C02514=1060.525,242.753,408.064,172.888,33.234,156.167
C02515=1060.519,242.505,408.092,172.886,33.230,156.166
C02516=1060.513,242.257,408.120,172.884,33.226,156.166
C02517=1060.506,242.008,408.148,172.881,33.222,156.165
C02518=1060.500,241.760,408.175,172.879,33.218,156.164
C02519=1060.494,241.512,408.204,172.877,33.215,156.163
C02520=1060.488,241.263,408.231,172.875,33.211,156.163
C02521=1060.481,241.015,408.258,172.872,33.207,156.162
C02522=1060.476,240.766,408.286,172.870,33.203,156.161
C02523=1060.469,240.518,408.314,172.868,33.200,156.161
C02524=1060.463,240.270,408.341,172.866,33.195,156.160
C02525=1060.457,240.021,408.369,172.863,33.192,156.159
C02526=1060.450,239.772,408.397,172.861,33.188,156.158
C02527=1060.444,239.524,408.424,172.859,33.184,156.158
C02528=1060.438,239.276,408.452,172.857,33.180,156.157
C02529=1060.432,239.028,408.480,172.854,33.176,156.156
C02530=1060.426,238.779,408.507,172.852,33.173,156.155
C02531=1060.419,238.530,408.534,172.850,33.169,156.155
C02532=1060.414,238.282,408.562,172.848,33.165,156.154
C02533=1060.408,238.033,408.589,172.845,33.161,156.153
C02534=1060.401,237.785,408.617,172.843,33.157,156.153
C02535=1060.395,237.537,408.645,172.841,33.153,156.152
C02536=1060.389,237.288,408.672,172.838,33.150,156.151
C02537=1060.383,237.040,408.699,172.835,33.146,156.150
C02538=1060.376,236.791,408.727,172.833,33.142,156.150
C02539=1060.371,236.543,408.754,172.831,33.138,156.149
C02540=1060.365,236.314,408.780,172.829,33.134,156.148
C02541=1060.359,236.084,408.805,172.827,33.131,156.148
C02542=1060.353,235.854,408.830,172.825,33.127,156.147
C02543=1060.348,235.624,408.856,172.823,33.124,156.146
C02544=1060.342,235.395,408.881,172.821,33.120,156.146
C02545=1060.336,235.165,408.906,172.819,33.117,156.145
C02546=1060.331,234.936,408.932,172.817,33.113,156.144
C02547=1060.325,234.706,408.956,172.815,33.109,156.143
C02548=1060.319,234.458,408.984,172.812,33.106,156.143
C02549=1060.313,234.209,409.011,172.810,33.101,156.142
C02550=1060.307,233.961,409.039,172.808,33.098,156.141
C02551=1060.301,233.712,409.066,172.806,33.094,156.141
C02552=1060.295,233.464,409.093,172.804,33.090,156.140
C02553=1060.289,233.215,409.120,172.801,33.086,156.139
C02554=1060.283,232.968,409.147,172.799,33.082,156.138
C02555=1060.276,232.718,409.174,172.797,33.078,156.138
C02556=1060.271,232.470,409.202,172.795,33.075,156.137
C02557=1060.264,232.221,409.229,172.793,33.071,156.136
C02558=1060.259,231.973,409.256,172.791,33.067,156.135
C02559=1060.252,231.725,409.284,172.788,33.063,156.135
C02560=1060.246,231.476,409.310,172.786,33.059,156.134
C02561=1060.240,231.228,409.338,172.784,33.055,156.133
C02562=1060.234,230.979,409.365,172.782,33.051,156.133
C02563=1060.228,230.731,409.391,172.780,33.047,156.132
C02564=1060.221,230.483,409.419,172.778,33.044,156.131
C02565=1060.216,230.234,409.446,172.775,33.040,156.130
C02566=1060.209,229.985,409.473,172.773,33.036,156.130
C02567=1060.203,229.737,409.500,172.771,33.032,156.129
C02568=1060.197,229.489,409.527,172.769,33.028,156.128
C02569=1060.191,229.240,409.554,172.767,33.024,156.127
C02570=1060.185,228.992,409.581,172.765,33.020,156.127
C02571=1060.179,228.743,409.608,172.762,33.017,156.126
C02572=1060.173,228.495,409.635,172.760,33.012,156.125
C02573=1060.166,228.246,409.661,172.758,33.009,156.125
C02574=1060.160,227.998,409.688,172.756,33.005,156.124
C02575=1060.153,227.749,409.715,172.754,33.001,156.123
C02576=1060.148,227.500,409.742,172.752,32.997,156.122
C02577=1060.142,227.252,409.768,172.750,32.993,156.122
C02578=1060.136,227.003,409.795,172.747,32.989,156.121
C02579=1060.129,226.755,409.822,172.745,32.985,156.120
C02580=1060.122,226.506,409.849,172.743,32.982,156.120
C02581=1060.117,226.258,409.876,172.741,32.978,156.119
C02582=1060.111,226.010,409.902,172.739,32.974,156.118
C02583=1060.104,225.761,409.929,172.737,32.970,156.117
C02584=1060.099,225.512,409.956,172.735,32.966,156.117
C02585=1060.092,225.264,409.982,172.732,32.962,156.116
C02586=1060.086,225.015,410.009,172.730,32.959,156.115
C02587=1060.080,224.767,410.036,172.728,32.954,156.114
C02588=1060.074,224.518,410.062,172.726,32.951,156.114
C02589=1060.068,224.269,410.089,172.724,32.946,156.113
C02590=1060.061,224.021,410.115,172.722,32.943,156.112
C02591=1060.056,223.773,410.142,172.720,32.939,156.112
C02592=1060.049,223.524,410.169,172.718,32.935,156.111
C02593=1060.043,223.276,410.196,172.716,32.931,156.110
C02594=1060.038,223.027,410.222,172.714,32.927,156.109
C02595=1060.031,222.779,410.248,172.711,32.923,156.109
C02596=1060.026,222.545,410.274,172.709,32.919,156.108
C02597=1060.020,222.312,410.299,172.708,32.916,156.107
C02598=1060.014,222.078,410.323,172.706,32.912,156.106
C02599=1060.009,221.845,410.348,172.704,32.909,156.106
C02600=1060.003,221.611,410.373,172.702,32.905,156.105
C02601=1059.997,221.378,410.398,172.700,32.901,156.104
C02602=1059.991,221.144,410.423,172.698,32.897,156.104
C02603=1059.985,220.910,410.448,172.696,32.893,156.103
C02604=1059.980,220.662,410.475,172.694,32.890,156.102
C02605=1059.973,220.414,410.501,172.692,32.886,156.102
C02606=1059.967,220.165,410.527,172.690,32.882,156.101
C02607=1059.960,219.916,410.554,172.687,32.878,156.100
C02608=1059.955,219.667,410.580,172.685,32.874,156.099
C02609=1059.948,219.419,410.606,172.683,32.870,156.099
C02610=1059.942,219.170,410.633,172.681,32.866,156.098
C02611=1059.935,218.922,410.659,172.679,32.863,156.097
C02612=1059.930,218.673,410.685,172.677,32.858,156.096
C02613=1059.923,218.425,410.711,172.675,32.855,156.096
C02614=1059.918,218.177,410.738,172.673,32.850,156.095
C02615=1059.911,217.927,410.764,172.671,32.847,156.094
C02616=1059.905,217.679,410.790,172.669,32.843,156.094
C02617=1059.899,217.431,410.817,172.667,32.839,156.093
C02618=1059.893,217.182,410.842,172.665,32.835,156.092
C02619=1059.887,216.933,410.869,172.663,32.831,156.091
C02620=1059.880,216.685,410.895,172.661,32.827,156.091
C02621=1059.875,216.436,410.921,172.659,32.823,156.090
C02622=1059.868,216.188,410.947,172.657,32.819,156.089
C02623=1059.862,215.940,410.974,172.655,32.815,156.088
C02624=1059.856,215.691,410.999,172.653,32.811,156.088
C02625=1059.850,215.442,411.026,172.651,32.808,156.087
C02626=1059.844,215.193,411.051,172.649,32.803,156.086
C02627=1059.838,214.945,411.078,172.647,32.800,156.085
C02628=1059.832,214.696,411.103,172.644,32.795,156.085
C02629=1059.826,214.448,411.130,172.642,32.792,156.084
C02630=1059.820,214.199,411.155,172.640,32.787,156.083
C02631=1059.814,213.951,411.182,172.638,32.784,156.083
C02632=1059.807,213.703,411.208,172.636,32.779,156.082
C02633=1059.800,213.453,411.234,172.634,32.776,156.081
C02634=1059.795,213.204,411.260,172.632,32.771,156.080
C02635=1059.788,212.956,411.286,172.630,32.768,156.080
C02636=1059.783,212.707,411.312,172.628,32.764,156.079
C02637=1059.777,212.459,411.338,172.626,32.760,156.078
C02638=1059.771,212.210,411.364,172.624,32.756,156.077
C02639=1059.765,211.962,411.390,172.622,32.752,156.077
C02640=1059.758,211.714,411.415,172.620,32.748,156.076
C02641=1059.753,211.465,411.441,172.618,32.744,156.075
C02642=1059.746,211.217,411.467,172.616,32.740,156.074
C02643=1059.740,210.967,411.493,172.614,32.736,156.074
C02644=1059.734,210.719,411.519,172.613,32.732,156.073
C02645=1059.728,210.470,411.545,172.611,32.728,156.072
C02646=1059.721,210.222,411.570,172.609,32.724,156.071
C02647=1059.715,209.974,411.596,172.607,32.720,156.071
C02648=1059.709,209.725,411.622,172.605,32.716,156.070
C02649=1059.703,209.476,411.647,172.604,32.712,156.069
C02650=1059.697,209.227,411.673,172.602,32.708,156.068
C02651=1059.690,208.979,411.699,172.600,32.704,156.068
C02652=1059.685,208.748,411.723,172.598,32.701,156.067
C02653=1059.679,208.517,411.746,172.596,32.697,156.066
C02654=1059.674,208.286,411.770,172.594,32.693,156.066
C02655=1059.668,208.055,411.794,172.592,32.689,156.065
C02656=1059.662,207.824,411.818,172.590,32.685,156.064
C02657=1059.656,207.592,411.842,172.589,32.682,156.063
C02658=1059.650,207.362,411.865,172.587,32.678,156.063
C02659=1059.645,207.130,411.889,172.585,32.674,156.062
C02660=1059.620,206.081,411.993,172.401,32.588,156.052
C02661=1059.614,205.833,412.019,172.399,32.585,156.052
C02662=1059.608,205.584,412.043,172.396,32.582,156.051
C02663=1059.602,205.335,412.068,172.394,32.579,156.051
C02664=1059.597,205.087,412.092,172.392,32.576,156.050
C02665=1059.591,204.837,412.117,172.389,32.573,156.050
C02666=1059.585,204.589,412.142,172.387,32.570,156.049
C02667=1059.579,204.340,412.166,172.386,32.567,156.049
C02668=1059.573,204.091,412.191,172.383,32.564,156.048
C02669=1059.567,203.843,412.216,172.381,32.560,156.047
C02670=1059.561,203.594,412.240,172.379,32.557,156.047
C02671=1059.556,203.345,412.264,172.376,32.554,156.046
C02672=1059.550,203.097,412.290,172.374,32.551,156.046
C02673=1059.544,202.848,412.314,172.372,32.548,156.045
C02674=1059.538,202.599,412.338,172.369,32.545,156.045
C02675=1059.532,202.351,412.363,172.367,32.542,156.044
C02676=1059.526,202.102,412.388,172.365,32.539,156.044
C02677=1059.521,201.853,412.412,172.362,32.536,156.043
C02678=1059.514,201.604,412.436,172.360,32.532,156.043
C02679=1059.508,201.356,412.461,172.358,32.530,156.042
C02680=1059.502,201.107,412.485,172.355,32.527,156.042
C02681=1059.496,200.858,412.510,172.353,32.523,156.041
C02682=1059.491,200.609,412.534,172.350,32.520,156.041
C02683=1059.484,200.360,412.558,172.348,32.518,156.040
C02684=1059.479,200.112,412.582,172.346,32.514,156.040
C02685=1059.472,199.863,412.606,172.344,32.511,156.039
C02686=1059.467,199.615,412.631,172.342,32.509,156.039
C02687=1059.460,199.366,412.655,172.340,32.506,156.038
C02688=1059.455,199.117,412.679,172.338,32.502,156.037
C02689=1059.448,198.868,412.703,172.335,32.500,156.037
C02690=1059.442,198.619,412.728,172.333,32.497,156.037
C02691=1059.437,198.370,412.752,172.331,32.493,156.036
C02692=1059.431,198.122,412.776,172.328,32.491,156.036
C02693=1059.425,197.873,412.801,172.326,32.488,156.035
C02694=1059.419,197.625,412.824,172.324,32.484,156.034
C02695=1059.413,197.375,412.849,172.321,32.482,156.034
C02696=1059.407,197.127,412.873,172.319,32.479,156.033
C02697=1059.401,196.878,412.897,172.317,32.475,156.033
C02698=1059.395,196.630,412.921,172.314,32.473,156.032
C02699=1059.389,196.380,412.945,172.312,32.470,156.032
C02700=1059.383,196.132,412.969,172.310,32.466,156.031
C02701=1059.377,195.883,412.994,172.309,32.464,156.031
C02702=1059.371,195.634,413.017,172.306,32.461,156.030
C02703=1059.366,195.386,413.042,172.304,32.457,156.030
C02704=1059.359,195.137,413.066,172.302,32.455,156.029
C02705=1059.354,194.888,413.090,172.299,32.452,156.029
C02706=1059.347,194.639,413.114,172.297,32.448,156.028
C02707=1059.342,194.391,413.138,172.295,32.446,156.028
C02708=1059.336,194.142,413.162,172.293,32.443,156.027
C02709=1059.330,193.892,413.186,172.290,32.439,156.027
C02710=1059.324,193.644,413.209,172.288,32.437,156.026
C02711=1059.318,193.395,413.234,172.286,32.434,156.026
C02712=1059.312,193.147,413.258,172.284,32.431,156.025
C02713=1059.307,192.898,413.282,172.281,32.428,156.025
C02714=1059.301,192.649,413.306,172.279,32.425,156.024
C02715=1059.296,192.400,413.330,172.277,32.422,156.024
C02716=1059.289,192.152,413.353,172.275,32.419,156.023
C02717=1059.283,191.903,413.377,172.273,32.416,156.023
C02718=1059.278,191.654,413.402,172.271,32.413,156.022
C02719=1059.272,191.406,413.425,172.269,32.410,156.022
C02720=1059.266,191.156,413.449,172.267,32.407,156.021
C02721=1059.260,190.873,413.476,172.264,32.404,156.021
C02722=1059.253,190.589,413.503,172.262,32.400,156.020
C02723=1059.246,190.306,413.531,172.259,32.397,156.020
C02724=1059.239,190.022,413.558,172.256,32.393,156.019
C02725=1059.234,189.773,413.582,172.254,32.391,156.019
C02726=1059.228,189.525,413.605,172.252,32.388,156.018
C02727=1059.222,189.275,413.629,172.250,32.384,156.017
C02728=1059.216,189.027,413.653,172.248,32.382,156.017
C02729=1059.210,188.778,413.677,172.245,32.379,156.016
C02730=1059.205,188.529,413.700,172.243,32.376,156.016
C02731=1059.199,188.280,413.724,172.242,32.373,156.016
C02732=1059.193,188.031,413.748,172.240,32.370,156.015
C02733=1059.188,187.783,413.771,172.238,32.367,156.015
C02734=1059.182,187.534,413.795,172.235,32.364,156.014
C02735=1059.176,187.284,413.819,172.233,32.361,156.014
C02736=1059.170,187.036,413.843,172.231,32.358,156.013
C02737=1059.165,186.788,413.867,172.229,32.355,156.012
C02738=1059.159,186.539,413.890,172.227,32.352,156.012
C02739=1059.153,186.290,413.914,172.224,32.349,156.011
C02740=1059.147,186.040,413.937,172.222,32.346,156.011
C02741=1059.141,185.792,413.961,172.220,32.343,156.011
C02742=1059.136,185.543,413.985,172.218,32.340,156.010
C02743=1059.130,185.295,414.008,172.216,32.338,156.010
C02744=1059.125,185.046,414.031,172.214,32.334,156.009
C02745=1059.119,184.797,414.055,172.212,32.332,156.009
C02746=1059.113,184.548,414.079,172.210,32.329,156.008
C02747=1059.107,184.299,414.102,172.208,32.325,156.007
C02748=1059.101,184.050,414.125,172.206,32.323,156.007
C02749=1059.095,183.802,414.148,172.204,32.320,156.007
C02750=1059.089,183.553,414.172,172.201,32.318,156.006
C02751=1059.083,183.304,414.195,172.199,32.314,156.006
C02752=1059.077,183.055,414.218,172.197,32.312,156.005
C02753=1059.071,182.806,414.242,172.195,32.309,156.005
C02754=1059.065,182.557,414.265,172.193,32.306,156.004
C02755=1059.059,182.308,414.288,172.190,32.303,156.004
C02756=1059.053,182.060,414.312,172.188,32.301,156.003
C02757=1059.047,181.810,414.335,172.186,32.298,156.003
C02758=1059.040,181.562,414.358,172.185,32.295,156.002
C02759=1059.034,181.313,414.381,172.183,32.292,156.002
C02760=1059.029,181.064,414.404,172.181,32.289,156.001
C02761=1059.023,180.815,414.427,172.178,32.287,156.001
C02762=1059.017,180.566,414.450,172.176,32.284,156.001
C02763=1059.011,180.318,414.474,172.174,32.281,156.000
C02764=1059.005,180.069,414.497,172.172,32.278,156.000
C02765=1058.999,179.820,414.520,172.170,32.276,155.999
C02766=1058.993,179.571,414.543,172.168,32.273,155.999
C02767=1058.987,179.322,414.567,172.165,32.270,155.998
C02768=1058.980,179.073,414.589,172.163,32.267,155.998
C02769=1058.974,178.824,414.612,172.161,32.265,155.997
C02770=1058.969,178.576,414.635,172.159,32.262,155.997
C02771=1058.963,178.327,414.658,172.158,32.259,155.996
C02772=1058.957,178.078,414.681,172.156,32.256,155.996
C02773=1058.952,177.829,414.704,172.154,32.254,155.996
C02774=1058.945,177.580,414.728,172.151,32.250,155.995
C02775=1058.938,177.331,414.750,172.149,32.248,155.995
C02776=1058.933,177.082,414.773,172.147,32.245,155.994
C02777=1058.927,176.833,414.796,172.145,32.242,155.994
C02778=1058.921,176.585,414.819,172.143,32.239,155.993
C02779=1058.916,176.336,414.842,172.141,32.237,155.993
C02780=1058.910,176.087,414.865,172.139,32.234,155.992
C02781=1058.904,175.838,414.888,172.137,32.231,155.992
C02782=1058.898,175.589,414.910,172.134,32.228,155.991
C02783=1058.891,175.340,414.934,172.132,32.226,155.991
C02784=1058.886,175.091,414.957,172.131,32.223,155.990
C02785=1058.879,174.808,414.983,172.129,32.220,155.990
C02786=1058.873,174.523,415.009,172.126,32.217,155.989
C02787=1058.866,174.239,415.035,172.124,32.213,155.989
C02788=1058.859,173.955,415.061,172.122,32.210,155.988
C02789=1058.853,173.706,415.084,172.119,32.208,155.988
C02790=1058.847,173.457,415.107,172.117,32.204,155.987
C02791=1058.841,173.208,415.129,172.115,32.202,155.987
C02792=1058.835,172.959,415.152,172.113,32.199,155.987
C02793=1058.829,172.710,415.175,172.111,32.196,155.986
C02794=1058.824,172.462,415.198,172.109,32.193,155.986
C02795=1058.818,172.213,415.221,172.108,32.191,155.985
C02796=1058.811,171.964,415.243,172.106,32.188,155.985
C02797=1058.806,171.715,415.266,172.104,32.185,155.984
C02798=1058.800,171.466,415.289,172.102,32.182,155.984
C02799=1058.794,171.217,415.312,172.100,32.180,155.983
C02800=1058.789,170.968,415.334,172.097,32.177,155.983
C02801=1058.782,170.719,415.357,172.095,32.174,155.982
C02802=1058.777,170.470,415.380,172.093,32.171,155.982
C02803=1058.771,170.222,415.403,172.091,32.169,155.981
C02804=1058.765,169.973,415.426,172.089,32.166,155.981
C02805=1058.759,169.724,415.449,172.087,32.163,155.980
C02806=1058.753,169.475,415.470,172.085,32.160,155.980
C02807=1058.748,169.226,415.493,172.084,32.157,155.980
C02808=1058.742,168.977,415.516,172.082,32.155,155.979
C02809=1058.737,168.729,415.539,172.080,32.152,155.979
C02810=1058.730,168.480,415.561,172.078,32.149,155.978
C02811=1058.725,168.230,415.583,172.076,32.146,155.978
C02812=1058.719,167.982,415.606,172.074,32.144,155.977
C02813=1058.713,167.733,415.629,172.072,32.141,155.977
C02814=1058.707,167.484,415.652,172.070,32.138,155.976
C02815=1058.701,167.235,415.674,172.068,32.135,155.976
C02816=1058.696,166.986,415.697,172.066,32.133,155.975
C02817=1058.690,166.737,415.720,172.063,32.129,155.975
C02818=1058.684,166.488,415.741,172.062,32.127,155.974
C02819=1058.679,166.239,415.764,172.060,32.124,155.974
C02820=1058.673,165.990,415.787,172.058,32.122,155.974
C02821=1058.667,165.742,415.810,172.056,32.118,155.973
C02822=1058.661,165.492,415.831,172.054,32.116,155.973
C02823=1058.655,165.243,415.854,172.052,32.113,155.972
C02824=1058.650,164.994,415.877,172.050,32.110,155.972
C02825=1058.645,164.746,415.899,172.048,32.107,155.971
C02826=1058.638,164.497,415.922,172.046,32.105,155.971
C02827=1058.633,164.248,415.944,172.044,32.102,155.970
C02828=1058.627,163.999,415.967,172.042,32.099,155.970
C02829=1058.621,163.750,415.989,172.041,32.096,155.969
C02830=1058.616,163.501,416.011,172.039,32.094,155.969
C02831=1058.610,163.252,416.034,172.037,32.091,155.968
C02832=1058.605,163.003,416.056,172.035,32.088,155.968
C02833=1058.598,162.754,416.078,172.033,32.085,155.968
C02834=1058.593,162.505,416.101,172.031,32.082,155.967
C02835=1058.588,162.257,416.123,172.029,32.080,155.967
C02836=1058.581,162.007,416.145,172.027,32.077,155.966
C02837=1058.576,161.759,416.168,172.025,32.074,155.966
C02838=1058.570,161.509,416.190,172.023,32.071,155.965
C02839=1058.564,161.261,416.212,172.021,32.069,155.965
C02840=1058.559,161.012,416.234,172.020,32.066,155.964
C02841=1058.553,160.763,416.257,172.018,32.063,155.964
C02842=1058.547,160.513,416.279,172.016,32.060,155.963
C02843=1058.541,160.265,416.301,172.014,32.058,155.963
C02844=1058.535,160.015,416.323,172.012,32.055,155.963
C02845=1058.530,159.767,416.345,172.010,32.052,155.962
C02846=1058.523,159.518,416.367,172.008,32.050,155.962
C02847=1058.518,159.269,416.389,172.006,32.047,155.961
C02848=1058.511,159.020,416.412,172.004,32.045,155.961
C02849=1058.505,158.735,416.437,172.002,32.041,155.960
C02850=1058.498,158.451,416.462,172.001,32.038,155.960
C02851=1058.491,158.167,416.486,171.998,32.035,155.959
C02852=1058.484,157.882,416.512,171.996,32.032,155.959
C02853=1058.479,157.633,416.534,171.994,32.030,155.958
C02854=1058.473,157.385,416.556,171.992,32.027,155.958
C02855=1058.467,157.136,416.578,171.990,32.024,155.958
C02856=1058.461,156.886,416.599,171.988,32.022,155.957
C02857=1058.456,156.638,416.621,171.986,32.019,155.957
C02858=1058.449,156.389,416.644,171.984,32.016,155.956
C02859=1058.443,156.140,416.665,171.982,32.013,155.956
C02860=1058.438,155.890,416.688,171.981,32.011,155.955
C02861=1058.432,155.642,416.709,171.979,32.008,155.955
C02862=1058.426,155.393,416.731,171.977,32.005,155.954
C02863=1058.420,155.144,416.753,171.975,32.003,155.954
C02864=1058.414,154.894,416.775,171.973,32.000,155.954
C02865=1058.409,154.646,416.796,171.971,31.998,155.953
C02866=1058.402,154.397,416.818,171.969,31.995,155.953
C02867=1058.396,154.148,416.840,171.967,31.992,155.952
C02868=1058.391,153.899,416.862,171.965,31.990,155.952
C02869=1058.385,153.650,416.884,171.963,31.987,155.952
C02870=1058.379,153.401,416.905,171.962,31.985,155.951
C02871=1058.373,153.152,416.927,171.961,31.982,155.951
C02872=1058.366,152.902,416.949,171.959,31.979,155.950
C02873=1058.362,152.654,416.971,171.957,31.976,155.950
C02874=1058.355,152.405,416.993,171.955,31.974,155.949
C02875=1058.349,152.156,417.015,171.953,31.971,155.949
C02876=1058.343,151.907,417.036,171.951,31.968,155.948
C02877=1058.337,151.658,417.057,171.949,31.966,155.948
C02878=1058.331,151.409,417.079,171.947,31.963,155.948
C02879=1058.326,151.160,417.101,171.945,31.961,155.947
C02880=1058.320,150.911,417.123,171.943,31.958,155.947
C02881=1058.314,150.662,417.144,171.942,31.955,155.946
C02882=1058.308,150.413,417.165,171.940,31.953,155.946
C02883=1058.302,150.164,417.187,171.938,31.950,155.945
C02884=1058.296,149.915,417.209,171.936,31.948,155.945
C02885=1058.291,149.666,417.230,171.934,31.945,155.945
C02886=1058.285,149.417,417.252,171.932,31.942,155.944
C02887=1058.279,149.168,417.274,171.930,31.940,155.944
C02888=1058.273,148.919,417.295,171.928,31.937,155.943
C02889=1058.267,148.670,417.317,171.927,31.935,155.943
C02890=1058.261,148.421,417.338,171.925,31.932,155.942
C02891=1058.255,148.172,417.360,171.924,31.929,155.942
C02892=1058.249,147.923,417.381,171.922,31.927,155.942
C02893=1058.243,147.674,417.403,171.920,31.924,155.941
C02894=1058.238,147.425,417.424,171.918,31.921,155.941
C02895=1058.232,147.175,417.445,171.916,31.919,155.940
C02896=1058.226,146.927,417.466,171.914,31.916,155.940
C02897=1058.220,146.678,417.488,171.912,31.914,155.939
C02898=1058.214,146.429,417.510,171.910,31.911,155.939
C02899=1058.208,146.180,417.531,171.908,31.908,155.939
C02900=1058.202,145.931,417.553,171.907,31.906,155.938
C02901=1058.196,145.682,417.574,171.905,31.903,155.938
C02902=1058.190,145.433,417.594,171.904,31.901,155.937
C02903=1058.184,145.184,417.616,171.902,31.898,155.937
C02904=1058.178,144.935,417.637,171.900,31.895,155.937
C02905=1058.172,144.686,417.659,171.898,31.893,155.936
C02906=1058.166,144.437,417.680,171.896,31.890,155.936
C02907=1058.161,144.188,417.701,171.894,31.888,155.935
C02908=1058.155,143.938,417.723,171.892,31.885,155.935
C02909=1058.149,143.690,417.744,171.890,31.882,155.934
C02910=1058.143,143.441,417.765,171.889,31.880,155.934
C02911=1058.137,143.191,417.787,171.887,31.877,155.934
C02912=1058.131,142.942,417.808,171.885,31.874,155.933
C02913=1058.124,142.658,417.832,171.883,31.872,155.933
C02914=1058.117,142.373,417.856,171.881,31.869,155.932
C02915=1058.111,142.088,417.881,171.879,31.866,155.932
C02916=1058.104,141.804,417.904,171.877,31.863,155.931
C02917=1058.098,141.555,417.926,171.875,31.860,155.931
C02918=1058.093,141.306,417.947,171.873,31.857,155.930
C02919=1058.087,141.056,417.968,171.872,31.855,155.930
C02920=1058.080,140.807,417.989,171.870,31.852,155.930
C02921=1058.074,140.559,418.010,171.868,31.850,155.929
C02922=1058.068,140.309,418.031,171.866,31.847,155.929
C02923=1058.063,140.060,418.053,171.865,31.844,155.928
C02924=1058.057,139.811,418.074,171.863,31.842,155.928
C02925=1058.051,139.562,418.095,171.861,31.839,155.927
C02926=1058.045,139.313,418.116,171.859,31.837,155.927
C02927=1058.039,139.064,418.136,171.857,31.834,155.927
C02928=1058.033,138.815,418.158,171.856,31.831,155.926
C02929=1058.028,138.566,418.179,171.854,31.829,155.926
C02930=1058.021,138.317,418.200,171.852,31.827,155.925
C02931=1058.015,138.068,418.221,171.851,31.824,155.925
C02932=1058.010,137.819,418.242,171.849,31.822,155.925
C02933=1058.003,137.570,418.262,171.847,31.819,155.924
C02934=1057.997,137.321,418.283,171.845,31.816,155.924
C02935=1057.992,137.072,418.305,171.843,31.814,155.923
C02936=1057.985,136.823,418.325,171.841,31.811,155.923
C02937=1057.980,136.574,418.346,171.840,31.808,155.922
C02938=1057.974,136.324,418.367,171.838,31.806,155.922
C02939=1057.968,136.076,418.388,171.837,31.803,155.922
C02940=1057.962,135.826,418.409,171.835,31.801,155.921
C02941=1057.956,135.577,418.429,171.833,31.799,155.921
C02942=1057.950,135.329,418.450,171.831,31.796,155.920
C02943=1057.944,135.079,418.471,171.829,31.793,155.920
C02944=1057.939,134.831,418.492,171.827,31.791,155.920
C02945=1057.932,134.581,418.512,171.825,31.788,155.919
C02946=1057.927,134.333,418.534,171.825,31.786,155.919
C02947=1057.921,134.083,418.555,171.823,31.783,155.918
C02948=1057.915,133.834,418.575,171.821,31.780,155.918
C02949=1057.909,133.585,418.596,171.819,31.778,155.917
C02950=1057.903,133.336,418.616,171.817,31.775,155.917
C02951=1057.897,133.087,418.638,171.815,31.772,155.917
C02952=1057.891,132.838,418.658,171.813,31.770,155.916
C02953=1057.885,132.589,418.678,171.812,31.768,155.916
C02954=1057.879,132.339,418.700,171.810,31.765,155.915
C02955=1057.874,132.090,418.721,171.809,31.763,155.915
C02956=1057.868,131.842,418.741,171.807,31.760,155.915
C02957=1057.862,131.592,418.762,171.805,31.757,155.914
C02958=1057.856,131.344,418.782,171.803,31.755,155.914
C02959=1057.849,131.094,418.802,171.801,31.752,155.913
C02960=1057.844,130.845,418.823,171.800,31.750,155.913
C02961=1057.837,130.596,418.844,171.798,31.748,155.913
C02962=1057.832,130.347,418.865,171.796,31.745,155.912
C02963=1057.826,130.098,418.885,171.794,31.742,155.912
C02964=1057.819,129.849,418.905,171.793,31.740,155.911
C02965=1057.813,129.600,418.926,171.791,31.738,155.911
C02966=1057.807,129.351,418.946,171.790,31.735,155.911
C02967=1057.801,129.102,418.966,171.788,31.732,155.910
C02968=1057.795,128.852,418.987,171.786,31.730,155.910
C02969=1057.789,128.603,419.007,171.784,31.728,155.910
C02970=1057.783,128.354,419.027,171.782,31.725,155.909
C02971=1057.777,128.105,419.049,171.780,31.723,155.909
C02972=1057.771,127.856,419.069,171.779,31.720,155.908
C02973=1057.764,127.607,419.089,171.778,31.717,155.908
C02974=1057.759,127.358,419.110,171.776,31.715,155.908
C02975=1057.753,127.109,419.130,171.774,31.713,155.907
C02976=1057.746,126.859,419.150,171.772,31.710,155.907
C02977=1057.740,126.575,419.173,171.770,31.707,155.906
C02978=1057.734,126.290,419.197,171.768,31.704,155.906
C02979=1057.726,126.005,419.220,171.766,31.702,155.905
C02980=1057.719,125.720,419.243,171.764,31.698,155.905
C02981=1057.713,125.471,419.263,171.763,31.696,155.904
C02982=1057.707,125.222,419.285,171.761,31.694,155.904
C02983=1057.701,124.973,419.305,171.759,31.691,155.904
C02984=1057.695,124.724,419.325,171.758,31.688,155.903
C02985=1057.689,124.475,419.345,171.756,31.686,155.903
C02986=1057.683,124.226,419.365,171.754,31.684,155.902
C02987=1057.677,123.976,419.386,171.752,31.681,155.902
C02988=1057.672,123.727,419.406,171.750,31.678,155.902
C02989=1057.666,123.478,419.426,171.749,31.676,155.901
C02990=1057.660,123.230,419.446,171.748,31.673,155.901
C02991=1057.653,122.980,419.466,171.746,31.671,155.900
C02992=1057.648,122.731,419.487,171.744,31.669,155.900
C02993=1057.642,122.482,419.507,171.742,31.666,155.900
C02994=1057.635,122.233,419.527,171.740,31.663,155.899
C02995=1057.630,121.984,419.548,171.739,31.661,155.899
C02996=1057.624,121.735,419.568,171.737,31.658,155.898
C02997=1057.618,121.486,419.588,171.735,31.656,155.898
C02998=1057.612,121.236,419.607,171.734,31.653,155.898
C02999=1057.606,120.987,419.628,171.732,31.651,155.897
C03000=1057.600,120.738,419.648,171.731,31.648,155.897
C03001=1057.594,120.489,419.668,171.729,31.646,155.896
C03002=1057.588,120.239,419.689,171.727,31.643,155.896
C03003=1057.582,119.990,419.709,171.725,31.640,155.896
C03004=1057.577,119.742,419.729,171.724,31.638,155.895
C03005=1057.571,119.493,419.749,171.722,31.635,155.895
C03006=1057.565,119.244,419.769,171.721,31.633,155.894
C03007=1057.559,118.994,419.790,171.719,31.631,155.894
C03008=1057.553,118.745,419.809,171.717,31.628,155.894
C03009=1057.547,118.496,419.829,171.716,31.625,155.893
C03010=1057.542,118.247,419.849,171.714,31.623,155.893
C03011=1057.536,117.998,419.869,171.712,31.620,155.892
C03012=1057.529,117.748,419.890,171.710,31.617,155.892
C03013=1057.523,117.499,419.909,171.708,31.615,155.892
C03014=1057.518,117.250,419.929,171.708,31.613,155.891
C03015=1057.512,117.001,419.949,171.706,31.610,155.891
C03016=1057.506,116.752,419.969,171.704,31.608,155.890
C03017=1057.500,116.503,419.989,171.702,31.605,155.890
C03018=1057.494,116.253,420.009,171.701,31.602,155.889
C03019=1057.489,116.004,420.029,171.699,31.600,155.889
C03020=1057.483,115.755,420.049,171.697,31.597,155.889
C03021=1057.477,115.507,420.069,171.695,31.595,155.888
C03022=1057.471,115.257,420.089,171.695,31.593,155.888
C03023=1057.466,115.008,420.109,171.693,31.590,155.887
C03024=1057.460,114.759,420.129,171.691,31.587,155.887
C03025=1057.454,114.510,420.149,171.689,31.585,155.887
C03026=1057.447,114.260,420.169,171.687,31.582,155.886
C03027=1057.441,114.011,420.189,171.686,31.579,155.886
C03028=1057.435,113.763,420.209,171.684,31.577,155.885
C03029=1057.430,113.513,420.228,171.682,31.575,155.885
C03030=1057.424,113.264,420.248,171.681,31.572,155.885
C03031=1057.418,113.016,420.268,171.680,31.570,155.884
C03032=1057.412,112.766,420.287,171.678,31.567,155.884
C03033=1057.406,112.517,420.307,171.676,31.564,155.883
C03034=1057.400,112.267,420.327,171.674,31.562,155.883
C03035=1057.394,112.018,420.347,171.673,31.560,155.883
C03036=1057.388,111.770,420.366,171.671,31.557,155.882
C03037=1057.382,111.520,420.386,171.669,31.554,155.882
C03038=1057.376,111.271,420.406,171.668,31.552,155.881
C03039=1057.370,111.022,420.425,171.666,31.550,155.881
C03040=1057.364,110.772,420.445,171.665,31.547,155.881
C03041=1057.357,110.487,420.467,171.663,31.545,155.880
C03042=1057.350,110.202,420.489,171.661,31.541,155.880
C03043=1057.344,109.918,420.512,171.659,31.539,155.879
C03044=1057.337,109.633,420.534,171.657,31.536,155.879
C03045=1057.331,109.384,420.554,171.656,31.533,155.878
C03046=1057.324,109.134,420.573,171.654,31.531,155.878
C03047=1057.318,108.885,420.593,171.652,31.529,155.878
C03048=1057.312,108.636,420.613,171.651,31.526,155.877
C03049=1057.307,108.386,420.632,171.649,31.523,155.877
C03050=1057.301,108.138,420.652,171.647,31.521,155.877
C03051=1057.295,107.888,420.671,171.645,31.519,155.876
C03052=1057.288,107.640,420.690,171.644,31.516,155.876
C03053=1057.282,107.390,420.710,171.643,31.514,155.875
C03054=1057.276,107.141,420.730,171.641,31.512,155.875
C03055=1057.271,106.892,420.749,171.639,31.509,155.875
C03056=1057.264,106.642,420.769,171.638,31.506,155.874
C03057=1057.258,106.393,420.788,171.636,31.504,155.874
C03058=1057.252,106.144,420.807,171.634,31.502,155.873
C03059=1057.246,105.895,420.827,171.632,31.499,155.873
C03060=1057.240,105.646,420.846,171.631,31.496,155.873
C03061=1057.235,105.396,420.866,171.630,31.494,155.872
C03062=1057.229,105.147,420.886,171.628,31.492,155.872
C03063=1057.222,104.898,420.904,171.626,31.489,155.871
C03064=1057.217,104.649,420.923,171.625,31.487,155.871
C03065=1057.211,104.400,420.943,171.623,31.484,155.871
C03066=1057.205,104.151,420.963,171.621,31.482,155.870
C03067=1057.198,103.901,420.981,171.619,31.479,155.870
C03068=1057.192,103.653,421.001,171.619,31.477,155.869
C03069=1057.187,103.403,421.020,171.617,31.474,155.869
C03070=1057.181,103.154,421.040,171.615,31.471,155.869
C03071=1057.175,102.905,421.060,171.613,31.469,155.868
C03072=1057.169,102.656,421.078,171.612,31.467,155.868
C03073=1057.163,102.406,421.098,171.610,31.464,155.868
C03074=1057.157,102.157,421.117,171.608,31.461,155.867
C03075=1057.151,101.908,421.137,171.606,31.459,155.867
C03076=1057.145,101.659,421.155,171.606,31.457,155.866
C03077=1057.139,101.410,421.175,171.604,31.454,155.866
C03078=1057.134,101.160,421.194,171.602,31.451,155.866
C03079=1057.128,100.911,421.214,171.601,31.449,155.865
C03080=1057.121,100.662,421.232,171.599,31.447,155.865
C03081=1057.115,100.413,421.252,171.597,31.444,155.864
C03082=1057.109,100.164,421.270,171.595,31.442,155.864
C03083=1057.103,99.914,421.290,171.595,31.440,155.864
C03084=1057.097,99.665,421.310,171.593,31.437,155.863
C03085=1057.091,99.416,421.328,171.591,31.434,155.863
C03086=1057.085,99.167,421.347,171.589,31.432,155.863
C03087=1057.079,98.918,421.366,171.588,31.430,155.862
C03088=1057.073,98.668,421.385,171.586,31.427,155.862
C03089=1057.067,98.419,421.404,171.584,31.425,155.861
C03090=1057.061,98.170,421.423,171.583,31.422,155.861
C03091=1057.055,97.921,421.442,171.582,31.420,155.861
C03092=1057.049,97.671,421.461,171.580,31.418,155.860
C03093=1057.042,97.423,421.481,171.578,31.415,155.860
C03094=1057.036,97.173,421.500,171.576,31.412,155.859
C03095=1057.030,96.924,421.518,171.575,31.410,155.859
C03096=1057.025,96.675,421.537,171.573,31.408,155.859
C03097=1057.019,96.426,421.557,171.571,31.405,155.858
C03098=1057.013,96.177,421.575,171.571,31.403,155.858
C03099=1057.007,95.927,421.594,171.569,31.401,155.858
C03100=1057.001,95.678,421.613,171.567,31.398,155.857
C03101=1056.995,95.429,421.632,171.565,31.395,155.857
C03102=1056.989,95.180,421.651,171.564,31.393,155.856
C03103=1056.983,94.930,421.670,171.562,31.391,155.856
C03104=1056.976,94.681,421.689,171.560,31.388,155.856
C03105=1056.970,94.396,421.711,171.559,31.385,155.855
C03106=1056.963,94.111,421.732,171.557,31.383,155.855
C03107=1056.956,93.827,421.753,171.555,31.379,155.854
C03108=1056.949,93.542,421.775,171.553,31.377,155.854
C03109=1056.944,93.292,421.794,171.552,31.374,155.853
C03110=1056.937,93.043,421.813,171.550,31.372,155.853
C03111=1056.931,92.794,421.832,171.548,31.369,155.853
C03112=1056.925,92.545,421.851,171.547,31.367,155.852
C03113=1056.919,92.295,421.870,171.546,31.364,155.852
C03114=1056.914,92.047,421.888,171.544,31.362,155.852
C03115=1056.908,91.797,421.907,171.542,31.359,155.851
C03116=1056.902,91.548,421.926,171.541,31.357,155.851
C03117=1056.895,91.298,421.944,171.539,31.355,155.850
C03118=1056.890,91.049,421.963,171.537,31.352,155.850
C03119=1056.883,90.800,421.982,171.536,31.350,155.850
C03120=1056.878,90.551,422.001,171.535,31.347,155.849
C03121=1056.872,90.302,422.020,171.533,31.345,155.849
C03122=1056.866,90.052,422.038,171.531,31.342,155.848
C03123=1056.860,89.803,422.057,171.530,31.340,155.848
C03124=1056.853,89.554,422.075,171.528,31.338,155.848
C03125=1056.847,89.305,422.094,171.526,31.335,155.847
C03126=1056.841,89.055,422.113,171.525,31.333,155.847
C03127=1056.835,88.805,422.131,171.524,31.330,155.847
C03128=1056.829,88.557,422.150,171.522,31.328,155.846
C03129=1056.823,88.308,422.168,171.520,31.326,155.846
C03130=1056.817,88.059,422.187,171.519,31.323,155.845
C03131=1056.810,87.809,422.205,171.517,31.321,155.845
C03132=1056.805,87.560,422.224,171.515,31.318,155.845
C03133=1056.798,87.310,422.243,171.514,31.316,155.844
C03134=1056.792,87.062,422.261,171.513,31.314,155.844
C03135=1056.786,86.812,422.279,171.511,31.311,155.844
C03136=1056.781,86.563,422.298,171.509,31.308,155.843
C03137=1056.774,86.314,422.317,171.508,31.306,155.843
C03138=1056.768,86.065,422.335,171.506,31.304,155.842
C03139=1056.762,85.815,422.353,171.504,31.301,155.842
C03140=1056.756,85.566,422.372,171.503,31.299,155.842
C03141=1056.750,85.317,422.391,171.502,31.296,155.841
C03142=1056.744,85.067,422.409,171.500,31.294,155.841
C03143=1056.738,84.818,422.427,171.498,31.292,155.841
C03144=1056.731,84.569,422.446,171.497,31.289,155.840
C03145=1056.726,84.320,422.464,171.495,31.287,155.840
C03146=1056.720,84.071,422.483,171.493,31.284,155.839
C03147=1056.714,83.821,422.501,171.492,31.282,155.839
C03148=1056.707,83.572,422.520,171.491,31.280,155.839
C03149=1056.702,83.323,422.538,171.489,31.277,155.838
C03150=1056.695,83.074,422.556,171.487,31.274,155.838
C03151=1056.690,82.824,422.575,171.486,31.273,155.838
C03152=1056.684,82.574,422.593,171.484,31.270,155.837
C03153=1056.678,82.326,422.611,171.483,31.267,155.837
C03154=1056.671,82.077,422.630,171.482,31.265,155.836
C03155=1056.665,81.827,422.648,171.480,31.263,155.836
C03156=1056.659,81.579,422.666,171.478,31.260,155.836
C03157=1056.654,81.329,422.685,171.476,31.258,155.835
C03158=1056.648,81.079,422.703,171.475,31.255,155.835
C03159=1056.642,80.830,422.721,171.473,31.253,155.835
C03160=1056.636,80.581,422.739,171.472,31.251,155.834
C03161=1056.630,80.332,422.757,171.471,31.248,155.834
C03162=1056.623,80.082,422.776,171.469,31.245,155.833
C03163=1056.618,79.833,422.794,171.467,31.243,155.833
C03164=1056.612,79.584,422.813,171.466,31.241,155.833
C03165=1056.606,79.334,422.831,171.464,31.238,155.832
C03166=1056.600,79.086,422.849,171.462,31.235,155.832
C03167=1056.594,78.836,422.867,171.461,31.233,155.832
C03168=1056.587,78.587,422.886,171.460,31.231,155.831
C03169=1056.581,78.302,422.906,171.458,31.228,155.831
C03170=1056.574,78.017,422.927,171.456,31.225,155.830
C03171=1056.567,77.731,422.948,171.454,31.223,155.830
C03172=1056.560,77.447,422.968,171.452,31.220,155.829
C03173=1056.554,77.198,422.987,171.451,31.217,155.829
C03174=1056.548,76.948,423.005,171.450,31.215,155.829
C03175=1056.542,76.699,423.022,171.448,31.213,155.828
C03176=1056.536,76.450,423.041,171.446,31.210,155.828
C03177=1056.530,76.200,423.059,171.444,31.208,155.828
C03178=1056.524,75.951,423.076,171.443,31.205,155.827
C03179=1056.518,75.702,423.095,171.441,31.203,155.827
C03180=1056.512,75.452,423.113,171.440,31.201,155.827
C03181=1056.505,75.203,423.130,171.439,31.198,155.826
C03182=1056.499,74.954,423.149,171.437,31.196,155.826
C03183=1056.493,74.705,423.167,171.435,31.193,155.825
C03184=1056.487,74.456,423.184,171.434,31.191,155.825
C03185=1056.481,74.206,423.203,171.432,31.189,155.825
C03186=1056.475,73.957,423.221,171.431,31.186,155.824
C03187=1056.469,73.708,423.238,171.429,31.184,155.824
C03188=1056.463,73.459,423.257,171.428,31.181,155.824
C03189=1056.457,73.209,423.275,171.426,31.179,155.823
C03190=1056.451,72.960,423.292,171.424,31.177,155.823
C03191=1056.445,72.710,423.310,171.423,31.174,155.822
C03192=1056.439,72.462,423.328,171.421,31.172,155.822
C03193=1056.432,72.212,423.346,171.420,31.169,155.822
C03194=1056.426,71.962,423.364,171.419,31.167,155.821
C03195=1056.421,71.713,423.382,171.417,31.165,155.821
C03196=1056.414,71.464,423.400,171.415,31.162,155.821
C03197=1056.409,71.215,423.418,171.413,31.160,155.820
C03198=1056.403,70.965,423.436,171.412,31.157,155.820
C03199=1056.396,70.716,423.453,171.411,31.155,155.819
C03200=1056.390,70.467,423.471,171.409,31.153,155.819
C03201=1056.384,70.217,423.489,171.408,31.150,155.819
C03202=1056.378,69.969,423.507,171.406,31.148,155.818
C03203=1056.372,69.719,423.525,171.404,31.145,155.818
C03204=1056.366,69.469,423.543,171.403,31.143,155.818
C03205=1056.360,69.221,423.560,171.401,31.141,155.817
C03206=1056.354,68.971,423.578,171.400,31.138,155.817
C03207=1056.348,68.722,423.595,171.399,31.136,155.817
C03208=1056.342,68.472,423.613,171.397,31.133,155.816
C03209=1056.336,68.223,423.630,171.395,31.131,155.816
C03210=1056.329,67.974,423.649,171.393,31.128,155.815
C03211=1056.323,67.724,423.667,171.392,31.127,155.815
C03212=1056.318,67.475,423.684,171.390,31.124,155.815
C03213=1056.311,67.226,423.702,171.389,31.121,155.814
C03214=1056.305,66.977,423.719,171.388,31.119,155.814
C03215=1056.299,66.727,423.737,171.386,31.116,155.814
C03216=1056.293,66.479,423.754,171.384,31.114,155.813
C03217=1056.287,66.229,423.772,171.383,31.112,155.813
C03218=1056.281,65.979,423.790,171.381,31.110,155.813
C03219=1056.275,65.730,423.807,171.380,31.107,155.812
C03220=1056.268,65.481,423.825,171.378,31.105,155.812
C03221=1056.263,65.232,423.842,171.377,31.102,155.811
C03222=1056.256,64.982,423.860,171.375,31.100,155.811
C03223=1056.251,64.733,423.877,171.373,31.098,155.811
C03224=1056.244,64.483,423.895,171.372,31.095,155.810
C03225=1056.238,64.235,423.912,171.371,31.093,155.810
C03226=1056.232,63.985,423.930,171.369,31.090,155.810
C03227=1056.226,63.736,423.947,171.368,31.088,155.809
C03228=1056.220,63.486,423.965,171.366,31.086,155.809
C03229=1056.213,63.238,423.982,171.364,31.084,155.809
C03230=1056.207,62.988,424.000,171.362,31.081,155.808
C03231=1056.201,62.738,424.017,171.361,31.079,155.808
C03232=1056.194,62.489,424.033,171.360,31.077,155.808
C03233=1056.187,62.204,424.054,171.358,31.074,155.807
C03234=1056.181,61.919,424.074,171.356,31.071,155.807
C03235=1056.173,61.634,424.094,171.354,31.069,155.806
C03236=1056.166,61.348,424.113,171.352,31.066,155.806
C03237=1056.160,61.099,424.131,171.350,31.064,155.806
C03238=1056.154,60.850,424.148,171.350,31.061,155.805
C03239=1056.147,60.600,424.166,171.348,31.059,155.805
C03240=1056.141,60.351,424.182,171.346,31.057,155.805
C03241=1056.135,60.101,424.200,171.345,31.055,155.804
C03242=1056.129,59.853,424.217,171.343,31.052,155.804
C03243=1056.123,59.603,424.235,171.341,31.050,155.804
C03244=1056.117,59.354,424.252,171.341,31.048,155.803
C03245=1056.110,59.104,424.268,171.339,31.045,155.803
C03246=1056.104,58.855,424.286,171.337,31.043,155.803
C03247=1056.098,58.606,424.303,171.335,31.040,155.802
C03248=1056.092,58.357,424.321,171.334,31.038,155.802
C03249=1056.086,58.107,424.337,171.332,31.036,155.801
C03250=1056.079,57.858,424.354,171.331,31.034,155.801
C03251=1056.074,57.609,424.372,171.330,31.031,155.801
C03252=1056.067,57.359,424.389,171.328,31.029,155.800
C03253=1056.062,57.110,424.406,171.326,31.026,155.800
C03254=1056.055,56.860,424.423,171.324,31.024,155.800
C03255=1056.049,56.612,424.440,171.323,31.022,155.799
C03256=1056.042,56.362,424.458,171.322,31.020,155.799
C03257=1056.036,56.112,424.475,171.320,31.017,155.799
C03258=1056.030,55.863,424.492,171.319,31.015,155.798
C03259=1056.024,55.614,424.510,171.317,31.013,155.798
C03260=1056.018,55.365,424.526,171.315,31.010,155.798
C03261=1056.012,55.115,424.544,171.314,31.008,155.797
C03262=1056.006,54.866,424.561,171.312,31.005,155.797
C03263=1055.999,54.616,424.577,171.311,31.003,155.797
C03264=1055.994,54.367,424.595,171.309,31.001,155.796
C03265=1055.987,54.118,424.612,171.308,30.999,155.796
C03266=1055.981,53.868,424.629,171.306,30.996,155.795
C03267=1055.975,53.619,424.646,171.304,30.994,155.795
C03268=1055.969,53.369,424.663,171.303,30.991,155.795
C03269=1055.963,53.121,424.680,171.302,30.989,155.794
C03270=1055.957,52.871,424.697,171.300,30.987,155.794
C03271=1055.951,52.621,424.714,171.299,30.985,155.794
C03272=1055.944,52.373,424.731,171.297,30.982,155.793
C03273=1055.939,52.123,424.748,171.295,30.980,155.793
C03274=1055.932,51.874,424.765,171.293,30.977,155.793
C03275=1055.927,51.624,424.782,171.293,30.975,155.792
C03276=1055.921,51.375,424.799,171.291,30.972,155.792
C03277=1055.914,51.126,424.816,171.289,30.970,155.792
C03278=1055.909,50.876,424.833,171.288,30.968,155.791
C03279=1055.902,50.627,424.850,171.286,30.966,155.791
C03280=1055.896,50.377,424.867,171.284,30.963,155.791
C03281=1055.890,50.129,424.884,171.283,30.961,155.790
C03282=1055.884,49.879,424.900,171.282,30.958,155.790
C03283=1055.878,49.630,424.918,171.280,30.956,155.790
C03284=1055.872,49.380,424.934,171.278,30.953,155.789
C03285=1055.866,49.131,424.952,171.277,30.951,155.789
C03286=1055.860,48.882,424.968,171.275,30.949,155.788
C03287=1055.853,48.632,424.985,171.274,30.947,155.788
C03288=1055.848,48.383,425.002,171.273,30.944,155.788
C03289=1055.842,48.133,425.018,171.271,30.942,155.787
C03290=1055.835,47.884,425.036,171.269,30.939,155.787
C03291=1055.830,47.634,425.053,171.267,30.937,155.787
C03292=1055.824,47.386,425.069,171.266,30.935,155.786
C03293=1055.818,47.136,425.086,171.265,30.933,155.786
C03294=1055.812,46.886,425.104,171.263,30.930,155.786
C03295=1055.806,46.637,425.120,171.262,30.928,155.785
C03296=1055.800,46.388,425.136,171.260,30.925,155.785
C03297=1055.793,46.103,425.156,171.258,30.922,155.784
C03298=1055.786,45.817,425.175,171.257,30.920,155.784
C03299=1055.779,45.532,425.195,171.255,30.917,155.784
C03300=1055.773,45.246,425.213,171.253,30.914,155.783
C03301=1055.766,44.997,425.230,171.252,30.912,155.783
C03302=1055.760,44.747,425.247,171.250,30.910,155.783
C03303=1055.755,44.498,425.263,171.248,30.908,155.782
C03304=1055.748,44.249,425.280,171.247,30.905,155.782
C03305=1055.742,44.000,425.297,171.246,30.903,155.782
C03306=1055.736,43.749,425.314,171.244,30.900,155.781
C03307=1055.730,43.501,425.331,171.242,30.898,155.781
C03308=1055.724,43.251,425.347,171.241,30.895,155.780
C03309=1055.718,43.002,425.363,171.239,30.893,155.780
C03310=1055.712,42.752,425.380,171.238,30.891,155.780
C03311=1055.706,42.503,425.397,171.236,30.889,155.779
C03312=1055.700,42.254,425.413,171.235,30.887,155.779
C03313=1055.694,42.004,425.429,171.233,30.884,155.779
C03314=1055.688,41.755,425.446,171.231,30.882,155.778
C03315=1055.681,41.506,425.463,171.230,30.879,155.778
C03316=1055.675,41.256,425.479,171.229,30.877,155.778
C03317=1055.669,41.007,425.496,171.227,30.875,155.777
C03318=1055.663,40.758,425.512,171.225,30.872,155.777
C03319=1055.656,40.507,425.528,171.224,30.870,155.777
C03320=1055.651,40.258,425.546,171.222,30.868,155.776
C03321=1055.645,40.009,425.562,171.220,30.865,155.776
C03322=1055.639,39.760,425.579,171.220,30.864,155.776
C03323=1055.633,39.510,425.595,171.218,30.861,155.775
C03324=1055.627,39.261,425.611,171.216,30.859,155.775
C03325=1055.621,39.011,425.628,171.214,30.856,155.775
C03326=1055.614,38.762,425.645,171.213,30.854,155.774
C03327=1055.608,38.513,425.661,171.211,30.852,155.774
C03328=1055.602,38.264,425.677,171.210,30.849,155.774
C03329=1055.596,38.014,425.693,171.209,30.847,155.773
C03330=1055.590,37.765,425.710,171.207,30.845,155.773
C03331=1055.584,37.515,425.726,171.205,30.842,155.773
C03332=1055.577,37.266,425.742,171.203,30.840,155.772
C03333=1055.571,37.016,425.758,171.203,30.838,155.772
C03334=1055.565,36.767,425.774,171.201,30.836,155.772
C03335=1055.559,36.518,425.791,171.199,30.833,155.771
C03336=1055.553,36.268,425.807,171.197,30.831,155.771
C03337=1055.547,36.018,425.824,171.196,30.829,155.771
C03338=1055.540,35.769,425.839,171.194,30.827,155.770
C03339=1055.534,35.520,425.856,171.193,30.825,155.770
C03340=1055.528,35.271,425.872,171.192,30.822,155.770
C03341=1055.522,35.022,425.889,171.190,30.820,155.769
C03342=1055.516,34.772,425.904,171.188,30.818,155.769
C03343=1055.510,34.522,425.921,171.186,30.815,155.769
C03344=1055.503,34.273,425.937,171.185,30.813,155.768
C03345=1055.497,34.023,425.953,171.184,30.811,155.768
C03346=1055.491,33.774,425.969,171.182,30.808,155.768
C03347=1055.485,33.525,425.985,171.180,30.806,155.767
C03348=1055.479,33.275,426.002,171.179,30.804,155.767
C03349=1055.473,33.026,426.017,171.177,30.801,155.767
C03350=1055.467,32.777,426.034,171.175,30.799,155.766
C03351=1055.460,32.527,426.050,171.175,30.797,155.766
C03352=1055.454,32.278,426.066,171.173,30.795,155.766
C03353=1055.448,32.028,426.083,171.171,30.793,155.765
C03354=1055.442,31.779,426.098,171.169,30.790,155.765
C03355=1055.436,31.530,426.115,171.168,30.788,155.765
C03356=1055.430,31.281,426.131,171.166,30.786,155.764
C03357=1055.424,31.031,426.147,171.165,30.784,155.764
C03358=1055.418,30.781,426.163,171.163,30.781,155.764
C03359=1055.411,30.532,426.178,171.162,30.779,155.763
C03360=1055.405,30.283,426.195,171.160,30.777,155.763
C03361=1055.399,29.997,426.213,171.158,30.774,155.763
C03362=1055.392,29.712,426.231,171.157,30.771,155.762
C03363=1055.384,29.426,426.250,171.155,30.769,155.762
C03364=1055.377,29.141,426.269,171.153,30.766,155.762
C03365=1055.371,28.891,426.284,171.151,30.764,155.761
C03366=1055.365,28.642,426.300,171.150,30.762,155.761
C03367=1055.359,28.392,426.316,171.149,30.760,155.761
C03368=1055.352,28.143,426.332,171.147,30.758,155.760
C03369=1055.346,27.894,426.348,171.145,30.755,155.760
C03370=1055.341,27.644,426.364,171.144,30.753,155.760
C03371=1055.334,27.395,426.379,171.142,30.751,155.759
C03372=1055.328,27.146,426.396,171.140,30.749,155.759
C03373=1055.322,26.896,426.412,171.139,30.746,155.759
C03374=1055.316,26.647,426.427,171.138,30.744,155.758
C03375=1055.310,26.397,426.443,171.136,30.742,155.758
C03376=1055.303,26.148,426.459,171.134,30.740,155.758
C03377=1055.297,25.898,426.474,171.132,30.737,155.757
C03378=1055.292,25.649,426.490,171.131,30.735,155.757
C03379=1055.285,25.400,426.506,171.130,30.733,155.757
C03380=1055.279,25.150,426.522,171.128,30.731,155.757
C03381=1055.273,24.901,426.537,171.126,30.729,155.756
C03382=1055.267,24.651,426.554,171.125,30.726,155.756
C03383=1055.260,24.402,426.569,171.123,30.724,155.756
C03384=1055.254,24.152,426.585,171.121,30.722,155.755
C03385=1055.248,23.903,426.600,171.120,30.720,155.755
C03386=1055.242,23.653,426.616,171.119,30.717,155.755
C03387=1055.236,23.404,426.632,171.117,30.715,155.754
C03388=1055.229,23.155,426.648,171.115,30.713,155.754
C03389=1055.224,22.905,426.663,171.113,30.711,155.754
C03390=1055.217,22.656,426.679,171.113,30.709,155.753
C03391=1055.211,22.406,426.695,171.111,30.706,155.753
C03392=1055.205,22.157,426.710,171.109,30.704,155.753
C03393=1055.199,21.908,426.727,171.107,30.702,155.752
C03394=1055.192,21.658,426.742,171.106,30.700,155.752
C03395=1055.186,21.409,426.758,171.104,30.697,155.752
C03396=1055.180,21.159,426.773,171.103,30.695,155.751
C03397=1055.174,20.910,426.789,171.101,30.693,155.751
C03398=1055.168,20.660,426.804,171.100,30.691,155.751
C03399=1055.162,20.411,426.820,171.098,30.689,155.751
C03400=1055.155,20.162,426.836,171.096,30.686,155.750
C03401=1055.149,19.912,426.851,171.095,30.684,155.750
C03402=1055.143,19.663,426.867,171.094,30.682,155.750
C03403=1055.137,19.413,426.883,171.092,30.680,155.749
C03404=1055.131,19.164,426.897,171.090,30.678,155.749
C03405=1055.125,18.914,426.913,171.088,30.675,155.749
C03406=1055.119,18.665,426.928,171.086,30.673,155.748
C03407=1055.112,18.416,426.944,171.086,30.671,155.748
C03408=1055.107,18.166,426.960,171.084,30.669,155.748
C03409=1055.100,17.917,426.975,171.082,30.666,155.747
C03410=1055.094,17.667,426.991,171.080,30.664,155.747
C03411=1055.087,17.418,427.006,171.079,30.662,155.747
C03412=1055.081,17.168,427.021,171.077,30.660,155.747
C03413=1055.075,16.918,427.037,171.076,30.658,155.746
C03414=1055.069,16.669,427.053,171.074,30.655,155.746
C03415=1055.062,16.419,427.068,171.073,30.653,155.746
C03416=1055.057,16.171,427.083,171.071,30.651,155.745
C03417=1055.051,15.921,427.098,171.069,30.649,155.745
C03418=1055.045,15.671,427.114,171.068,30.647,155.745
C03419=1055.038,15.422,427.130,171.066,30.644,155.744
C03420=1055.032,15.172,427.145,171.065,30.642,155.744
C03421=1055.026,14.923,427.161,171.063,30.640,155.744
C03422=1055.020,14.673,427.176,171.061,30.638,155.743
C03423=1055.013,14.424,427.191,171.059,30.636,155.743
C03424=1055.008,14.174,427.206,171.059,30.634,155.743
C03425=1055.001,13.891,427.224,171.057,30.631,155.742
C03426=1054.993,13.606,427.241,171.055,30.629,155.742
C03427=1054.986,13.322,427.258,171.053,30.626,155.742
C03428=1054.979,13.038,427.276,171.050,30.624,155.742
C03429=1054.973,12.788,427.291,171.050,30.622,155.741
C03430=1054.966,12.539,427.306,171.048,30.620,155.741
C03431=1054.960,12.289,427.321,171.046,30.618,155.741
C03432=1054.953,12.040,427.336,171.044,30.616,155.740
C03433=1054.947,11.791,427.351,171.043,30.614,155.740
C03434=1054.942,11.541,427.367,171.041,30.612,155.740
C03435=1054.935,11.291,427.381,171.040,30.609,155.740
C03436=1054.929,11.042,427.397,171.038,30.607,155.739
C03437=1054.922,10.793,427.412,171.036,30.605,155.739
C03438=1054.916,10.543,427.427,171.035,30.603,155.739
C03439=1054.910,10.293,427.442,171.033,30.601,155.738
C03440=1054.904,10.044,427.457,171.032,30.599,155.738
C03441=1054.898,9.795,427.472,171.030,30.597,155.738
C03442=1054.891,9.545,427.488,171.028,30.595,155.738
C03443=1054.885,9.296,427.503,171.027,30.593,155.737
C03444=1054.879,9.046,427.518,171.025,30.590,155.737
C03445=1054.873,8.797,427.532,171.023,30.588,155.737
C03446=1054.867,8.548,427.547,171.022,30.586,155.736
C03447=1054.860,8.298,427.562,171.020,30.584,155.736
C03448=1054.854,8.048,427.577,171.019,30.582,155.736
C03449=1054.847,7.799,427.593,171.017,30.580,155.735
C03450=1054.842,7.550,427.608,171.015,30.578,155.735
C03451=1054.836,7.300,427.623,171.014,30.576,155.735
C03452=1054.829,7.051,427.638,171.012,30.574,155.735
C03453=1054.823,6.801,427.653,171.011,30.572,155.734
C03454=1054.817,6.551,427.668,171.009,30.569,155.734
C03455=1054.811,6.302,427.682,171.007,30.567,155.734
C03456=1054.804,6.053,427.697,171.005,30.565,155.733
C03457=1054.798,5.803,427.712,171.004,30.562,155.733
C03458=1054.792,5.553,427.727,171.003,30.560,155.733
C03459=1054.786,5.304,427.742,171.001,30.558,155.733
C03460=1054.779,5.055,427.757,170.999,30.556,155.732
C03461=1054.774,4.805,427.772,170.997,30.554,155.732
C03462=1054.768,4.556,427.787,170.996,30.552,155.732
C03463=1054.762,4.306,427.802,170.995,30.550,155.731
C03464=1054.755,4.057,427.817,170.993,30.548,155.731
C03465=1054.749,3.807,427.832,170.991,30.546,155.731
C03466=1054.743,3.558,427.846,170.989,30.543,155.731
C03467=1054.737,3.308,427.861,170.987,30.541,155.730
C03468=1054.730,3.059,427.876,170.987,30.539,155.730
C03469=1054.724,2.810,427.891,170.985,30.537,155.730
C03470=1054.718,2.560,427.906,170.983,30.535,155.729
C03471=1054.712,2.310,427.921,170.981,30.533,155.729
C03472=1054.706,2.061,427.935,170.979,30.531,155.729
C03473=1054.700,1.812,427.950,170.978,30.529,155.729
C03474=1054.693,1.562,427.965,170.977,30.527,155.728
C03475=1054.687,1.313,427.980,170.975,30.524,155.728
C03476=1054.681,1.063,427.995,170.973,30.522,155.728
C03477=1054.675,0.813,428.010,170.971,30.520,155.727
C03478=1054.670,0.564,428.024,170.969,30.518,155.727
C03479=1054.664,0.314,428.039,170.969,30.516,155.727
C03480=1054.657,0.065,428.054,170.967,30.514,155.727
C03481=1054.651,-0.184,428.068,170.965,30.512,155.726
C03482=1054.645,-0.434,428.083,170.963,30.510,155.726
C03483=1054.639,-0.684,428.098,170.961,30.508,155.726
C03484=1054.633,-0.933,428.113,170.960,30.505,155.725
C03485=1054.627,-1.183,428.127,170.959,30.503,155.725
C03486=1054.621,-1.432,428.142,170.957,30.501,155.725
C03487=1054.615,-1.682,428.157,170.955,30.499,155.725
C03488=1054.608,-1.931,428.172,170.953,30.497,155.724
C03489=1054.601,-2.213,428.188,170.951,30.495,155.724
C03490=1054.595,-2.495,428.205,170.950,30.493,155.724
C03491=1054.588,-2.778,428.221,170.948,30.490,155.723
C03492=1054.581,-3.060,428.237,170.946,30.488,155.723
C03493=1054.574,-3.310,428.252,170.944,30.486,155.723
C03494=1054.568,-3.559,428.267,170.942,30.483,155.722
C03495=1054.562,-3.809,428.281,170.941,30.481,155.722
C03496=1054.557,-4.058,428.295,170.940,30.479,155.722
C03497=1054.550,-4.308,428.310,170.938,30.478,155.722
C03498=1054.543,-4.557,428.325,170.936,30.476,155.721
C03499=1054.538,-4.806,428.339,170.934,30.473,155.721
C03500=1054.531,-5.056,428.354,170.933,30.471,155.721
C03501=1054.524,-5.305,428.368,170.931,30.469,155.721
C03502=1054.519,-5.555,428.382,170.930,30.468,155.720
C03503=1054.512,-5.805,428.397,170.928,30.466,155.720
C03504=1054.506,-6.054,428.411,170.926,30.464,155.720
C03505=1054.500,-6.304,428.425,170.924,30.461,155.720
C03506=1054.493,-6.553,428.440,170.923,30.459,155.719
C03507=1054.487,-6.802,428.454,170.921,30.458,155.719
C03508=1054.481,-7.053,428.469,170.919,30.456,155.719
C03509=1054.475,-7.301,428.483,170.918,30.454,155.719
C03510=1054.469,-7.551,428.497,170.916,30.451,155.718
C03511=1054.462,-7.801,428.512,170.915,30.449,155.718
C03512=1054.456,-8.050,428.526,170.913,30.448,155.718
C03513=1054.450,-8.300,428.540,170.911,30.446,155.718
C03514=1054.444,-8.549,428.555,170.909,30.443,155.717
C03515=1054.437,-8.799,428.568,170.907,30.441,155.717
C03516=1054.431,-9.048,428.583,170.906,30.439,155.717
C03517=1054.425,-9.298,428.597,170.905,30.438,155.717
C03518=1054.420,-9.547,428.612,170.903,30.436,155.716
C03519=1054.413,-9.797,428.625,170.901,30.433,155.716
C03520=1054.407,-10.046,428.640,170.899,30.431,155.716
C03521=1054.401,-10.296,428.655,170.897,30.429,155.715
C03522=1054.394,-10.545,428.668,170.896,30.428,155.715
C03523=1054.388,-10.795,428.683,170.895,30.426,155.715
C03524=1054.383,-11.044,428.697,170.893,30.423,155.715
C03525=1054.375,-11.294,428.711,170.891,30.421,155.714
C03526=1054.370,-11.543,428.725,170.889,30.420,155.714
C03527=1054.364,-11.793,428.739,170.887,30.418,155.714
C03528=1054.357,-12.042,428.753,170.886,30.415,155.714
C03529=1054.351,-12.292,428.768,170.884,30.413,155.713
C03530=1054.345,-12.541,428.782,170.882,30.411,155.713
C03531=1054.339,-12.791,428.796,170.881,30.410,155.713
C03532=1054.333,-13.040,428.810,170.879,30.408,155.713
C03533=1054.327,-13.290,428.825,170.878,30.405,155.712
C03534=1054.320,-13.539,428.839,170.876,30.403,155.712
C03535=1054.314,-13.789,428.853,170.874,30.402,155.712
C03536=1054.309,-14.039,428.867,170.872,30.400,155.712
C03537=1054.302,-14.288,428.881,170.870,30.397,155.711
C03538=1054.296,-14.538,428.895,170.869,30.395,155.711
C03539=1054.290,-14.787,428.909,170.868,30.394,155.711
C03540=1054.284,-15.037,428.923,170.866,30.392,155.711
C03541=1054.278,-15.286,428.937,170.864,30.390,155.710
C03542=1054.271,-15.536,428.951,170.862,30.387,155.710
C03543=1054.265,-15.785,428.965,170.860,30.386,155.710
C03544=1054.259,-16.035,428.979,170.859,30.384,155.710
C03545=1054.253,-16.284,428.993,170.857,30.382,155.709
C03546=1054.246,-16.534,429.007,170.855,30.380,155.709
C03547=1054.240,-16.783,429.020,170.854,30.378,155.709
C03548=1054.234,-17.034,429.035,170.852,30.376,155.709
C03549=1054.227,-17.282,429.049,170.850,30.374,155.708
C03550=1054.221,-17.533,429.063,170.849,30.372,155.708
C03551=1054.215,-17.782,429.076,170.847,30.371,155.708
C03552=1054.209,-18.031,429.091,170.845,30.368,155.708
C03553=1054.201,-18.312,429.106,170.843,30.366,155.707
C03554=1054.195,-18.593,429.121,170.841,30.364,155.707
C03555=1054.188,-18.873,429.137,170.840,30.362,155.707
C03556=1054.181,-19.154,429.152,170.838,30.360,155.707
C03557=1054.175,-19.404,429.166,170.836,30.358,155.706
C03558=1054.168,-19.653,429.180,170.834,30.356,155.706
C03559=1054.162,-19.902,429.194,170.832,30.354,155.706
C03560=1054.156,-20.152,429.208,170.831,30.352,155.706
C03561=1054.149,-20.402,429.221,170.829,30.350,155.705
C03562=1054.144,-20.651,429.235,170.827,30.349,155.705
C03563=1054.137,-20.901,429.249,170.825,30.346,155.705
C03564=1054.131,-21.150,429.262,170.823,30.345,155.705
C03565=1054.125,-21.399,429.276,170.821,30.343,155.705
C03566=1054.118,-21.649,429.290,170.821,30.341,155.704
C03567=1054.113,-21.899,429.304,170.819,30.339,155.704
C03568=1054.106,-22.149,429.317,170.817,30.337,155.704
C03569=1054.100,-22.398,429.331,170.815,30.335,155.704
C03570=1054.094,-22.647,429.345,170.813,30.333,155.703
C03571=1054.087,-22.897,429.359,170.811,30.332,155.703
C03572=1054.082,-23.147,429.373,170.810,30.330,155.703
C03573=1054.076,-23.396,429.386,170.808,30.327,155.703
C03574=1054.069,-23.646,429.400,170.806,30.326,155.703
C03575=1054.063,-23.896,429.414,170.804,30.324,155.702
C03576=1054.057,-24.145,429.427,170.802,30.322,155.702
C03577=1054.051,-24.394,429.440,170.802,30.320,155.702
C03578=1054.045,-24.644,429.454,170.800,30.319,155.702
C03579=1054.039,-24.894,429.468,170.798,30.316,155.701
C03580=1054.032,-25.143,429.481,170.796,30.314,155.701
C03581=1054.026,-25.393,429.495,170.794,30.313,155.701
C03582=1054.020,-25.642,429.508,170.792,30.311,155.701
C03583=1054.015,-25.892,429.522,170.791,30.309,155.701
C03584=1054.008,-26.141,429.536,170.789,30.307,155.700
C03585=1054.002,-26.391,429.549,170.787,30.305,155.700
C03586=1053.996,-26.641,429.563,170.785,30.303,155.700
C03587=1053.990,-26.890,429.576,170.783,30.302,155.700
C03588=1053.983,-27.140,429.590,170.782,30.299,155.699
C03589=1053.977,-27.389,429.603,170.780,30.298,155.699
C03590=1053.971,-27.639,429.616,170.779,30.296,155.699
C03591=1053.964,-27.888,429.630,170.777,30.294,155.699
C03592=1053.958,-28.138,429.644,170.775,30.293,155.699
C03593=1053.952,-28.387,429.657,170.773,30.291,155.698
C03594=1053.946,-28.637,429.671,170.772,30.289,155.698
C03595=1053.939,-28.887,429.684,170.770,30.287,155.698
C03596=1053.933,-29.136,429.697,170.768,30.285,155.698
C03597=1053.927,-29.386,429.710,170.766,30.284,155.698
C03598=1053.921,-29.635,429.723,170.764,30.282,155.697
C03599=1053.914,-29.885,429.737,170.762,30.280,155.697
C03600=1053.908,-30.134,429.751,170.761,30.278,155.697
C03601=1053.902,-30.384,429.764,170.759,30.276,155.697
C03602=1053.895,-30.634,429.778,170.757,30.275,155.697
C03603=1053.890,-30.884,429.790,170.755,30.273,155.696
C03604=1053.883,-31.133,429.803,170.753,30.271,155.696
C03605=1053.877,-31.382,429.817,170.752,30.269,155.696
C03606=1053.871,-31.631,429.830,170.750,30.267,155.696
C03607=1053.864,-31.881,429.844,170.748,30.266,155.695
C03608=1053.858,-32.131,429.857,170.747,30.264,155.695
C03609=1053.852,-32.381,429.869,170.745,30.262,155.695
C03610=1053.846,-32.630,429.883,170.743,30.261,155.695
C03611=1053.840,-32.879,429.897,170.742,30.258,155.695
C03612=1053.833,-33.129,429.910,170.740,30.257,155.694
C03613=1053.828,-33.379,429.923,170.738,30.255,155.694
C03614=1053.821,-33.628,429.936,170.736,30.253,155.694
C03615=1053.815,-33.878,429.949,170.734,30.252,155.694
C03616=1053.809,-34.127,429.963,170.733,30.249,155.694
C03617=1053.802,-34.407,429.977,170.731,30.248,155.693
C03618=1053.795,-34.687,429.992,170.729,30.246,155.693
C03619=1053.788,-34.967,430.007,170.726,30.243,155.693
C03620=1053.781,-35.247,430.021,170.724,30.242,155.693
C03621=1053.774,-35.497,430.035,170.722,30.240,155.693
C03622=1053.768,-35.746,430.048,170.721,30.238,155.692
C03623=1053.762,-35.996,430.061,170.719,30.236,155.692
C03624=1053.756,-36.245,430.074,170.717,30.234,155.692
C03625=1053.750,-36.495,430.087,170.715,30.233,155.692
C03626=1053.745,-36.744,430.100,170.713,30.231,155.692
C03627=1053.739,-36.994,430.113,170.712,30.230,155.691
C03628=1053.733,-37.244,430.126,170.710,30.227,155.691
C03629=1053.726,-37.494,430.140,170.708,30.226,155.691
C03630=1053.720,-37.743,430.153,170.707,30.224,155.691
C03631=1053.714,-37.993,430.166,170.705,30.222,155.690
C03632=1053.707,-38.242,430.179,170.703,30.221,155.690
C03633=1053.701,-38.492,430.192,170.702,30.219,155.690
C03634=1053.695,-38.741,430.205,170.700,30.217,155.690
C03635=1053.689,-38.991,430.217,170.698,30.215,155.690
C03636=1053.682,-39.240,430.230,170.696,30.214,155.690
C03637=1053.677,-39.490,430.243,170.694,30.212,155.689
C03638=1053.670,-39.740,430.256,170.692,30.211,155.689
C03639=1053.664,-39.990,430.269,170.691,30.209,155.689
C03640=1053.658,-40.239,430.282,170.689,30.207,155.689
